LIN {X 0,Y 290.88,Z 169.752,A -85,B 0,C 180,E1 -16935.017,E2 -16935.017} C_VEL
LIN {X 0,Y 287.972,Z 170.097,A -85,B 0,C 180,E1 -16936.892,E2 -16936.892} C_VEL
LIN {X 0,Y 285.493,Z 170.39,A -85,B 0,C 180,E1 -16938.414,E2 -16938.414} C_VEL
LIN {X 0,Y 284.452,Z 170.52,A -85,B 0,C 180,E1 -16939.596,E2 -16939.596} C_VEL
LIN {X 0,Y 284.382,Z 170.533,A -85,B 0,C 180,E1 -16939.996,E2 -16939.996} C_VEL
LIN {X 0,Y 284.369,Z 170.558,A -85,B 0,C 180,E1 -16943.876,E2 -16943.876} C_VEL
LIN {X 0,Y 284.395,Z 170.53,A -85,B 0,C 180,E1 -16947.174,E2 -16947.174} C_VEL
LIN {X 0,Y 284.293,Z 170.571,A -85,B 0,C 180,E1 -16951.275,E2 -16951.275} C_VEL
LIN {X 0,Y 284.341,Z 170.55,A -85,B 0,C 180,E1 -16955.349,E2 -16955.349} C_VEL
LIN {X 0,Y 284.319,Z 170.568,A -85,B 0,C 180,E1 -16958.169,E2 -16958.169} C_VEL
LIN {X 0,Y 284.27,Z 170.574,A -85,B 0,C 180,E1 -16962.125,E2 -16962.125} C_VEL
LIN {X 0,Y 284.257,Z 170.577,A -85,B 0,C 180,E1 -16966.19,E2 -16966.19} C_VEL
LIN {X 0,Y 284.309,Z 170.539,A -85,B 0,C 180,E1 -16970.025,E2 -16970.025} C_VEL
LIN {X 0,Y 284.377,Z 170.673,A -85,B 0,C 180,E1 -16973.511,E2 -16973.511} C_VEL
LIN {X 0,Y 286.09,Z 178.895,A -85,B 0,C 180,E1 -16977.286,E2 -16977.286} C_VEL
LIN {X 0,Y 287.859,Z 188.158,A -85,B 0,C 180,E1 -16981.346,E2 -16981.346} C_VEL
LIN {X 0,Y 288.12,Z 189.357,A -85,B 0,C 180,E1 -16981.632,E2 -16981.632} C_VEL
LIN {X 0,Y 290.426,Z 195.694,A -85,B 0,C 180,E1 -16982.073,E2 -16982.073} C_VEL
LIN {X 0,Y 295.176,Z 217.529,A -85,B 0,C 180,E1 -16983.141,E2 -16983.141} C_VEL
LIN {X 0,Y 298.276,Z 235.786,A -85,B 0,C 180,E1 -16983.919,E2 -16983.919} C_VEL
LIN {X 0,Y 296.617,Z 295.017,A -85,B 0,C 180,E1 -16985.364,E2 -16985.364} C_VEL
LIN {X 0,Y 295.946,Z 305.327,A -85,B 0,C 180,E1 -16985.771,E2 -16985.771} C_VEL
LIN {X 0,Y 295.071,Z 314.839,A -85,B 0,C 180,E1 -16986.302,E2 -16986.302} C_VEL
LIN {X 0,Y 293.886,Z 324.916,A -85,B 0,C 180,E1 -16987.04,E2 -16987.04} C_VEL
LIN {X 0,Y 292.65,Z 334.674,A -85,B 0,C 180,E1 -16987.961,E2 -16987.961} C_VEL
LIN {X 0,Y 291.052,Z 344.737,A -85,B 0,C 180,E1 -16989.135,E2 -16989.135} C_VEL
LIN {X 0,Y 289.074,Z 356.234,A -85,B 0,C 180,E1 -16990.84,E2 -16990.84} C_VEL
LIN {X 0,Y 287.646,Z 364.301,A -85,B 0,C 180,E1 -16992.343,E2 -16992.343} C_VEL
LIN {X 0,Y 286.356,Z 371.575,A -85,B 0,C 180,E1 -16993.972,E2 -16993.972} C_VEL
LIN {X 0,Y 285.164,Z 378.112,A -85,B 0,C 180,E1 -16995.732,E2 -16995.732} C_VEL
LIN {X 0,Y 284.291,Z 382.612,A -85,B 0,C 180,E1 -16997.145,E2 -16997.145} C_VEL
LIN {X 0,Y 283.419,Z 388.106,A -85,B 0,C 180,E1 -16999.282,E2 -16999.282} C_VEL
LIN {X 0,Y 282.805,Z 392.433,A -85,B 0,C 180,E1 -17001.425,E2 -17001.425} C_VEL
LIN {X 0,Y 282.557,Z 394.802,A -85,B 0,C 180,E1 -17002.856,E2 -17002.856} C_VEL
LIN {X 0,Y 282.364,Z 397.026,A -85,B 0,C 180,E1 -17004.626,E2 -17004.626} C_VEL
LIN {X 0,Y 282.338,Z 399.054,A -85,B 0,C 180,E1 -17007.146,E2 -17007.146} C_VEL
LIN {X 0,Y 282.332,Z 399.644,A -85,B 0,C 180,E1 -17008.574,E2 -17008.574} C_VEL
LIN {X 0,Y 282.332,Z 399.644,A -85,B 0,C 180,E1 -17011.426,E2 -17011.426} C_VEL
LIN {X 0,Y 282.337,Z 399.054,A -85,B 0,C 180,E1 -17012.854,E2 -17012.854} C_VEL
LIN {X 0,Y 282.387,Z 396.602,A -85,B 0,C 180,E1 -17015.713,E2 -17015.713} C_VEL
LIN {X 0,Y 282.676,Z 393.651,A -85,B 0,C 180,E1 -17017.859,E2 -17017.859} C_VEL
LIN {X 0,Y 283.172,Z 389.66,A -85,B 0,C 180,E1 -17020.005,E2 -17020.005} C_VEL
LIN {X 0,Y 283.96,Z 384.528,A -85,B 0,C 180,E1 -17022.144,E2 -17022.144} C_VEL
LIN {X 0,Y 284.958,Z 379.268,A -85,B 0,C 180,E1 -17023.914,E2 -17023.914} C_VEL
LIN {X 0,Y 286.097,Z 372.951,A -85,B 0,C 180,E1 -17025.677,E2 -17025.677} C_VEL
LIN {X 0,Y 287.263,Z 367.002,A -85,B 0,C 180,E1 -17027.073,E2 -17027.073} C_VEL
LIN {X 0,Y 288.4,Z 360.072,A -85,B 0,C 180,E1 -17028.469,E2 -17028.469} C_VEL
LIN {X 0,Y 289.832,Z 351.895,A -85,B 0,C 180,E1 -17029.845,E2 -17029.845} C_VEL
LIN {X 0,Y 291.276,Z 343.386,A -85,B 0,C 180,E1 -17031.033,E2 -17031.033} C_VEL
LIN {X 0,Y 292.597,Z 334.673,A -85,B 0,C 180,E1 -17032.043,E2 -17032.043} C_VEL
LIN {X 0,Y 293.956,Z 324.918,A -85,B 0,C 180,E1 -17032.955,E2 -17032.955} C_VEL
LIN {X 0,Y 295.044,Z 314.838,A -85,B 0,C 180,E1 -17033.701,E2 -17033.701} C_VEL
LIN {X 0,Y 295.936,Z 305.326,A -85,B 0,C 180,E1 -17034.23,E2 -17034.23} C_VEL
LIN {X 0,Y 296.643,Z 295.017,A -85,B 0,C 180,E1 -17034.634,E2 -17034.634} C_VEL
LIN {X 0,Y 298.183,Z 234.871,A -85,B 0,C 180,E1 -17036.113,E2 -17036.113} C_VEL
LIN {X 0,Y 294.305,Z 213.339,A -85,B 0,C 180,E1 -17037.056,E2 -17037.056} C_VEL
LIN {X 0,Y 290.089,Z 194.522,A -85,B 0,C 180,E1 -17037.994,E2 -17037.994} C_VEL
LIN {X 0,Y 288.05,Z 189.055,A -85,B 0,C 180,E1 -17038.402,E2 -17038.402} C_VEL
LIN {X 0,Y 287.273,Z 184.811,A -85,B 0,C 180,E1 -17040.1,E2 -17040.1} C_VEL
LIN {X 0,Y 285.624,Z 176.503,A -85,B 0,C 180,E1 -17043.786,E2 -17043.786} C_VEL
LIN {X 0,Y 284.366,Z 170.578,A -85,B 0,C 180,E1 -17046.601,E2 -17046.601} C_VEL
LIN {X 0,Y 284.308,Z 170.539,A -85,B 0,C 180,E1 -17049.994,E2 -17049.994} C_VEL
LIN {X 0,Y 284.247,Z 170.575,A -85,B 0,C 180,E1 -17054.19,E2 -17054.19} C_VEL
LIN {X 0,Y 284.273,Z 170.574,A -85,B 0,C 180,E1 -17058.124,E2 -17058.124} C_VEL
LIN {X 0,Y 284.327,Z 170.567,A -85,B 0,C 180,E1 -17062.276,E2 -17062.276} C_VEL
LIN {X 0,Y 284.308,Z 170.548,A -85,B 0,C 180,E1 -17065.35,E2 -17065.35} C_VEL
LIN {X 0,Y 284.293,Z 170.571,A -85,B 0,C 180,E1 -17068.725,E2 -17068.725} C_VEL
LIN {X 0,Y 284.395,Z 170.53,A -85,B 0,C 180,E1 -17072.826,E2 -17072.826} C_VEL
LIN {X 0,Y 284.366,Z 170.561,A -85,B 0,C 180,E1 -17076.706,E2 -17076.706} C_VEL
LIN {X 0,Y 284.401,Z 170.521,A -85,B 0,C 180,E1 -17081.261,E2 -17081.261} C_VEL
LIN {X 0,Y 284.491,Z 170.539,A -85,B 0,C 180,E1 -17084.458,E2 -17084.458} C_VEL
LIN {X 0,Y 284.486,Z 170.522,A -85,B 0,C 180,E1 -17088.601,E2 -17088.601} C_VEL
LIN {X 0,Y 284.637,Z 170.496,A -85,B 0,C 180,E1 -17091.48,E2 -17091.48} C_VEL
LIN {X 0,Y 284.596,Z 170.532,A -85,B 0,C 180,E1 -17094.33,E2 -17094.33} C_VEL
LIN {X 0,Y 284.852,Z 170.475,A -85,B 0,C 180,E1 -17098.585,E2 -17098.585} C_VEL
LIN {X 0,Y 284.853,Z 170.47,A -85,B 0,C 180,E1 -17101.413,E2 -17101.413} C_VEL
LIN {X 0,Y 284.696,Z 170.513,A -85,B 0,C 180,E1 -17107.089,E2 -17107.089} C_VEL
LIN {X 0,Y 284.563,Z 170.5,A -85,B 0,C 180,E1 -17109.955,E2 -17109.955} C_VEL
LIN {X 0,Y 284.478,Z 170.55,A -85,B 0,C 180,E1 -17114.302,E2 -17114.302} C_VEL
LIN {X 0,Y 284.422,Z 170.536,A -85,B 0,C 180,E1 -17117.248,E2 -17117.248} C_VEL
LIN {X 0,Y 284.375,Z 170.533,A -85,B 0,C 180,E1 -17120.242,E2 -17120.242} C_VEL
LIN {X 0,Y 284.366,Z 170.563,A -85,B 0,C 180,E1 -17123.875,E2 -17123.875} C_VEL
LIN {X 0,Y 284.393,Z 170.531,A -85,B 0,C 180,E1 -17127.173,E2 -17127.173} C_VEL
LIN {X 0,Y 284.292,Z 170.575,A -85,B 0,C 180,E1 -17131.274,E2 -17131.274} C_VEL
LIN {X 0,Y 284.357,Z 170.544,A -85,B 0,C 180,E1 -17135.353,E2 -17135.353} C_VEL
LIN {X 0,Y 284.319,Z 170.569,A -85,B 0,C 180,E1 -17138.167,E2 -17138.167} C_VEL
LIN {X 0,Y 284.265,Z 170.569,A -85,B 0,C 180,E1 -17142.124,E2 -17142.124} C_VEL
LIN {X 0,Y 284.264,Z 170.535,A -85,B 0,C 180,E1 -17146.191,E2 -17146.191} C_VEL
LIN {X 0,Y 284.303,Z 170.538,A -85,B 0,C 180,E1 -17150.024,E2 -17150.024} C_VEL
LIN {X 0,Y 284.346,Z 170.546,A -85,B 0,C 180,E1 -17153.617,E2 -17153.617} C_VEL
LIN {X 0,Y 284.305,Z 170.553,A -85,B 0,C 180,E1 -17157.189,E2 -17157.189} C_VEL
LIN {X 0,Y 284.362,Z 170.704,A -85,B 0,C 180,E1 -17160.852,E2 -17160.852} C_VEL
LIN {X 0,Y 284.575,Z 171.612,A -85,B 0,C 180,E1 -17161.125,E2 -17161.125} C_VEL
LIN {X 0,Y 292.693,Z 186.861,A -85,B 0,C 180,E1 -17162.447,E2 -17162.447} C_VEL
LIN {X 0,Y 300.723,Z 198.195,A -85,B 0,C 180,E1 -17163.545,E2 -17163.545} C_VEL
LIN {X 0,Y 308.771,Z 207.249,A -85,B 0,C 180,E1 -17164.599,E2 -17164.599} C_VEL
LIN {X 0,Y 315.653,Z 214.555,A -85,B 0,C 180,E1 -17165.617,E2 -17165.617} C_VEL
LIN {X 0,Y 321.435,Z 220.417,A -85,B 0,C 180,E1 -17166.56,E2 -17166.56} C_VEL
LIN {X 0,Y 328.774,Z 227.475,A -85,B 0,C 180,E1 -17167.909,E2 -17167.909} C_VEL
LIN {X 0,Y 335.567,Z 233.937,A -85,B 0,C 180,E1 -17169.296,E2 -17169.296} C_VEL
LIN {X 0,Y 343.566,Z 240.897,A -85,B 0,C 180,E1 -17171.056,E2 -17171.056} C_VEL
LIN {X 0,Y 349.047,Z 245.344,A -85,B 0,C 180,E1 -17172.381,E2 -17172.381} C_VEL
LIN {X 0,Y 354.863,Z 250.07,A -85,B 0,C 180,E1 -17173.931,E2 -17173.931} C_VEL
LIN {X 0,Y 359.024,Z 253.254,A -85,B 0,C 180,E1 -17175.137,E2 -17175.137} C_VEL
LIN {X 0,Y 364.017,Z 257.245,A -85,B 0,C 180,E1 -17176.739,E2 -17176.739} C_VEL
LIN {X 0,Y 368.789,Z 260.213,A -85,B 0,C 180,E1 -17178.465,E2 -17178.465} C_VEL
LIN {X 0,Y 370.688,Z 261.609,A -85,B 0,C 180,E1 -17179.248,E2 -17179.248} C_VEL
LIN {X 0,Y 374.455,Z 264.816,A -85,B 0,C 180,E1 -17181.025,E2 -17181.025} C_VEL
LIN {X 0,Y 377.636,Z 266.924,A -85,B 0,C 180,E1 -17182.836,E2 -17182.836} C_VEL
LIN {X 0,Y 380.183,Z 268.235,A -85,B 0,C 180,E1 -17184.697,E2 -17184.697} C_VEL
LIN {X 0,Y 381.337,Z 268.729,A -85,B 0,C 180,E1 -17185.772,E2 -17185.772} C_VEL
LIN {X 0,Y 382.556,Z 269.148,A -85,B 0,C 180,E1 -17187.355,E2 -17187.355} C_VEL
LIN {X 0,Y 383.208,Z 269.566,A -85,B 0,C 180,E1 -17188.949,E2 -17188.949} C_VEL
LIN {X 0,Y 383.351,Z 269.507,A -85,B 0,C 180,E1 -17190,E2 -17190} C_VEL
LIN {X 0,Y 383.05,Z 269.43,A -85,B 0,C 180,E1 -17191.577,E2 -17191.577} C_VEL
LIN {X 0,Y 382.228,Z 268.951,A -85,B 0,C 180,E1 -17193.162,E2 -17193.162} C_VEL
LIN {X 0,Y 380.501,Z 268.419,A -85,B 0,C 180,E1 -17195.024,E2 -17195.024} C_VEL
LIN {X 0,Y 377.945,Z 267.115,A -85,B 0,C 180,E1 -17196.961,E2 -17196.961} C_VEL
LIN {X 0,Y 374.474,Z 264.83,A -85,B 0,C 180,E1 -17198.966,E2 -17198.966} C_VEL
LIN {X 0,Y 370.839,Z 261.73,A -85,B 0,C 180,E1 -17200.689,E2 -17200.689} C_VEL
LIN {X 0,Y 368.619,Z 260.105,A -85,B 0,C 180,E1 -17201.604,E2 -17201.604} C_VEL
LIN {X 0,Y 364.035,Z 257.251,A -85,B 0,C 180,E1 -17203.255,E2 -17203.255} C_VEL
LIN {X 0,Y 359.029,Z 253.234,A -85,B 0,C 180,E1 -17204.863,E2 -17204.863} C_VEL
LIN {X 0,Y 353.786,Z 249.277,A -85,B 0,C 180,E1 -17206.371,E2 -17206.371} C_VEL
LIN {X 0,Y 348.293,Z 244.643,A -85,B 0,C 180,E1 -17207.809,E2 -17207.809} C_VEL
LIN {X 0,Y 341.138,Z 238.842,A -85,B 0,C 180,E1 -17209.493,E2 -17209.493} C_VEL
LIN {X 0,Y 335.159,Z 233.574,A -85,B 0,C 180,E1 -17210.79,E2 -17210.79} C_VEL
LIN {X 0,Y 329.509,Z 228.106,A -85,B 0,C 180,E1 -17211.947,E2 -17211.947} C_VEL
LIN {X 0,Y 322.949,Z 221.914,A -85,B 0,C 180,E1 -17213.17,E2 -17213.17} C_VEL
LIN {X 0,Y 316.392,Z 215.413,A -85,B 0,C 180,E1 -17214.263,E2 -17214.263} C_VEL
LIN {X 0,Y 308.197,Z 206.704,A -85,B 0,C 180,E1 -17215.476,E2 -17215.476} C_VEL
LIN {X 0,Y 299.593,Z 196.708,A -85,B 0,C 180,E1 -17216.602,E2 -17216.602} C_VEL
LIN {X 0,Y 292.262,Z 186.12,A -85,B 0,C 180,E1 -17217.618,E2 -17217.618} C_VEL
LIN {X 0,Y 284.576,Z 171.61,A -85,B 0,C 180,E1 -17218.876,E2 -17218.876} C_VEL
LIN {X 0,Y 284.353,Z 170.626,A -85,B 0,C 180,E1 -17219.19,E2 -17219.19} C_VEL
LIN {X 0,Y 284.303,Z 170.551,A -85,B 0,C 180,E1 -17222.945,E2 -17222.945} C_VEL
LIN {X 0,Y 284.346,Z 170.546,A -85,B 0,C 180,E1 -17226.383,E2 -17226.383} C_VEL
LIN {X 0,Y 284.302,Z 170.537,A -85,B 0,C 180,E1 -17229.995,E2 -17229.995} C_VEL
LIN {X 0,Y 284.261,Z 170.543,A -85,B 0,C 180,E1 -17234.195,E2 -17234.195} C_VEL
LIN {X 0,Y 284.268,Z 170.565,A -85,B 0,C 180,E1 -17238.125,E2 -17238.125} C_VEL
LIN {X 0,Y 284.331,Z 170.57,A -85,B 0,C 180,E1 -17242.275,E2 -17242.275} C_VEL
LIN {X 0,Y 284.319,Z 170.544,A -85,B 0,C 180,E1 -17245.353,E2 -17245.353} C_VEL
LIN {X 0,Y 284.292,Z 170.575,A -85,B 0,C 180,E1 -17248.726,E2 -17248.726} C_VEL
LIN {X 0,Y 284.393,Z 170.531,A -85,B 0,C 180,E1 -17252.827,E2 -17252.827} C_VEL
LIN {X 0,Y 284.363,Z 170.563,A -85,B 0,C 180,E1 -17256.708,E2 -17256.708} C_VEL
LIN {X 0,Y 284.399,Z 170.523,A -85,B 0,C 180,E1 -17261.262,E2 -17261.262} C_VEL
LIN {X 0,Y 284.489,Z 170.547,A -85,B 0,C 180,E1 -17264.46,E2 -17264.46} C_VEL
LIN {X 0,Y 284.485,Z 170.522,A -85,B 0,C 180,E1 -17268.602,E2 -17268.602} C_VEL
LIN {X 0,Y 284.657,Z 170.498,A -85,B 0,C 180,E1 -17271.482,E2 -17271.482} C_VEL
LIN {X 0,Y 284.599,Z 170.534,A -85,B 0,C 180,E1 -17274.332,E2 -17274.332} C_VEL
LIN {X 0,Y 284.853,Z 170.47,A -85,B 0,C 180,E1 -17278.587,E2 -17278.587} C_VEL
LIN {X 0,Y 284.852,Z 170.475,A -85,B 0,C 180,E1 -17281.415,E2 -17281.415} C_VEL
LIN {X 0,Y 284.685,Z 170.508,A -85,B 0,C 180,E1 -17287.091,E2 -17287.091} C_VEL
LIN {X 0,Y 284.517,Z 170.505,A -85,B 0,C 180,E1 -17289.958,E2 -17289.958} C_VEL
LIN {X 0,Y 284.48,Z 170.545,A -85,B 0,C 180,E1 -17294.304,E2 -17294.304} C_VEL
LIN {X 0,Y 284.424,Z 170.529,A -85,B 0,C 180,E1 -17297.249,E2 -17297.249} C_VEL
LIN {X 0,Y 284.382,Z 170.533,A -85,B 0,C 180,E1 -17299.996,E2 -17299.996} C_VEL
LIN {X 0,Y 283.743,Z 170.628,A -85,B 0,C 180,E1 -17301.179,E2 -17301.179} C_VEL
LIN {X 0,Y 280.866,Z 170.999,A -85,B 0,C 180,E1 -17303.104,E2 -17303.104} C_VEL
LIN {X 0,Y 278.415,Z 171.293,A -85,B 0,C 180,E1 -17304.669,E2 -17304.669} C_VEL
LIN {X 0,Y 277.379,Z 171.409,A -85,B 0,C 180,E1 -17305.882,E2 -17305.882} C_VEL
LIN {X 0,Y 277.306,Z 171.414,A -85,B 0,C 180,E1 -17306.293,E2 -17306.293} C_VEL
LIN {X 0,Y 277.272,Z 171.447,A -85,B 0,C 180,E1 -17310.482,E2 -17310.482} C_VEL
LIN {X 0,Y 277.247,Z 171.426,A -85,B 0,C 180,E1 -17313.897,E2 -17313.897} C_VEL
LIN {X 0,Y 277.272,Z 171.447,A -85,B 0,C 180,E1 -17317.469,E2 -17317.469} C_VEL
LIN {X 0,Y 277.21,Z 171.445,A -85,B 0,C 180,E1 -17321.237,E2 -17321.237} C_VEL
LIN {X 0,Y 277.202,Z 171.447,A -85,B 0,C 180,E1 -17325.227,E2 -17325.227} C_VEL
LIN {X 0,Y 277.224,Z 171.421,A -85,B 0,C 180,E1 -17329.513,E2 -17329.513} C_VEL
LIN {X 0,Y 277.359,Z 171.598,A -85,B 0,C 180,E1 -17332.962,E2 -17332.962} C_VEL
LIN {X 0,Y 278.83,Z 178.676,A -85,B 0,C 180,E1 -17336.323,E2 -17336.323} C_VEL
LIN {X 0,Y 280.375,Z 186.527,A -85,B 0,C 180,E1 -17339.912,E2 -17339.912} C_VEL
LIN {X 0,Y 280.83,Z 188.826,A -85,B 0,C 180,E1 -17340.795,E2 -17340.795} C_VEL
LIN {X 0,Y 284.482,Z 198.321,A -85,B 0,C 180,E1 -17341.516,E2 -17341.516} C_VEL
LIN {X 0,Y 289.64,Z 223.006,A -85,B 0,C 180,E1 -17342.739,E2 -17342.739} C_VEL
LIN {X 0,Y 291.878,Z 236.965,A -85,B 0,C 180,E1 -17343.34,E2 -17343.34} C_VEL
LIN {X 0,Y 290.182,Z 294.832,A -85,B 0,C 180,E1 -17344.779,E2 -17344.779} C_VEL
LIN {X 0,Y 289.491,Z 305.135,A -85,B 0,C 180,E1 -17345.195,E2 -17345.195} C_VEL
LIN {X 0,Y 288.568,Z 314.647,A -85,B 0,C 180,E1 -17345.734,E2 -17345.734} C_VEL
LIN {X 0,Y 287.513,Z 323.719,A -85,B 0,C 180,E1 -17346.405,E2 -17346.405} C_VEL
LIN {X 0,Y 286.342,Z 332.852,A -85,B 0,C 180,E1 -17347.259,E2 -17347.259} C_VEL
LIN {X 0,Y 284.897,Z 341.844,A -85,B 0,C 180,E1 -17348.283,E2 -17348.283} C_VEL
LIN {X 0,Y 283.35,Z 350.568,A -85,B 0,C 180,E1 -17349.492,E2 -17349.492} C_VEL
LIN {X 0,Y 281.978,Z 357.96,A -85,B 0,C 180,E1 -17350.717,E2 -17350.717} C_VEL
LIN {X 0,Y 280.525,Z 366.236,A -85,B 0,C 180,E1 -17352.372,E2 -17352.372} C_VEL
LIN {X 0,Y 279.224,Z 372.758,A -85,B 0,C 180,E1 -17353.927,E2 -17353.927} C_VEL
LIN {X 0,Y 278.022,Z 379.075,A -85,B 0,C 180,E1 -17355.732,E2 -17355.732} C_VEL
LIN {X 0,Y 276.983,Z 384.336,A -85,B 0,C 180,E1 -17357.545,E2 -17357.545} C_VEL
LIN {X 0,Y 276.164,Z 389.468,A -85,B 0,C 180,E1 -17359.739,E2 -17359.739} C_VEL
LIN {X 0,Y 275.606,Z 393.458,A -85,B 0,C 180,E1 -17361.938,E2 -17361.938} C_VEL
LIN {X 0,Y 275.256,Z 397.09,A -85,B 0,C 180,E1 -17364.736,E2 -17364.736} C_VEL
LIN {X 0,Y 275.247,Z 398.862,A -85,B 0,C 180,E1 -17367.073,E2 -17367.073} C_VEL
LIN {X 0,Y 275.256,Z 399.453,A -85,B 0,C 180,E1 -17368.537,E2 -17368.537} C_VEL
LIN {X 0,Y 275.256,Z 399.453,A -85,B 0,C 180,E1 -17371.463,E2 -17371.463} C_VEL
LIN {X 0,Y 275.246,Z 398.862,A -85,B 0,C 180,E1 -17372.927,E2 -17372.927} C_VEL
LIN {X 0,Y 275.3,Z 396.41,A -85,B 0,C 180,E1 -17375.861,E2 -17375.861} C_VEL
LIN {X 0,Y 275.606,Z 393.458,A -85,B 0,C 180,E1 -17378.062,E2 -17378.062} C_VEL
LIN {X 0,Y 276.164,Z 389.468,A -85,B 0,C 180,E1 -17380.261,E2 -17380.261} C_VEL
LIN {X 0,Y 276.983,Z 384.336,A -85,B 0,C 180,E1 -17382.455,E2 -17382.455} C_VEL
LIN {X 0,Y 278.023,Z 379.075,A -85,B 0,C 180,E1 -17384.268,E2 -17384.268} C_VEL
LIN {X 0,Y 279.228,Z 372.758,A -85,B 0,C 180,E1 -17386.073,E2 -17386.073} C_VEL
LIN {X 0,Y 280.666,Z 365.808,A -85,B 0,C 180,E1 -17387.718,E2 -17387.718} C_VEL
LIN {X 0,Y 281.662,Z 359.88,A -85,B 0,C 180,E1 -17388.927,E2 -17388.927} C_VEL
LIN {X 0,Y 283.143,Z 351.702,A -85,B 0,C 180,E1 -17390.334,E2 -17390.334} C_VEL
LIN {X 0,Y 284.645,Z 343.194,A -85,B 0,C 180,E1 -17391.547,E2 -17391.547} C_VEL
LIN {X 0,Y 286.011,Z 334.481,A -85,B 0,C 180,E1 -17392.578,E2 -17392.578} C_VEL
LIN {X 0,Y 287.44,Z 324.727,A -85,B 0,C 180,E1 -17393.506,E2 -17393.506} C_VEL
LIN {X 0,Y 288.542,Z 314.646,A -85,B 0,C 180,E1 -17394.269,E2 -17394.269} C_VEL
LIN {X 0,Y 289.488,Z 305.135,A -85,B 0,C 180,E1 -17394.805,E2 -17394.805} C_VEL
LIN {X 0,Y 290.206,Z 294.826,A -85,B 0,C 180,E1 -17395.218,E2 -17395.218} C_VEL
LIN {X 0,Y 291.804,Z 235.968,A -85,B 0,C 180,E1 -17396.694,E2 -17396.694} C_VEL
LIN {X 0,Y 288.25,Z 215.924,A -85,B 0,C 180,E1 -17397.597,E2 -17397.597} C_VEL
LIN {X 0,Y 284.205,Z 197.401,A -85,B 0,C 180,E1 -17398.54,E2 -17398.54} C_VEL
LIN {X 0,Y 280.826,Z 188.828,A -85,B 0,C 180,E1 -17399.203,E2 -17399.203} C_VEL
LIN {X 0,Y 280.112,Z 185.125,A -85,B 0,C 180,E1 -17400.726,E2 -17400.726} C_VEL
LIN {X 0,Y 278.412,Z 176.684,A -85,B 0,C 180,E1 -17404.607,E2 -17404.607} C_VEL
LIN {X 0,Y 277.34,Z 171.483,A -85,B 0,C 180,E1 -17407.144,E2 -17407.144} C_VEL
LIN {X 0,Y 277.211,Z 171.427,A -85,B 0,C 180,E1 -17411.236,E2 -17411.236} C_VEL
LIN {X 0,Y 277.202,Z 171.446,A -85,B 0,C 180,E1 -17415.226,E2 -17415.226} C_VEL
LIN {X 0,Y 277.223,Z 171.438,A -85,B 0,C 180,E1 -17419.511,E2 -17419.511} C_VEL
LIN {X 0,Y 277.272,Z 171.447,A -85,B 0,C 180,E1 -17422.531,E2 -17422.531} C_VEL
LIN {X 0,Y 277.247,Z 171.426,A -85,B 0,C 180,E1 -17426.103,E2 -17426.103} C_VEL
LIN {X 0,Y 277.261,Z 171.448,A -85,B 0,C 180,E1 -17429.538,E2 -17429.538} C_VEL
LIN {X 0,Y 277.356,Z 171.406,A -85,B 0,C 180,E1 -17432.863,E2 -17432.863} C_VEL
LIN {X 0,Y 277.328,Z 171.435,A -85,B 0,C 180,E1 -17436.079,E2 -17436.079} C_VEL
LIN {X 0,Y 277.343,Z 171.401,A -85,B 0,C 180,E1 -17440.765,E2 -17440.765} C_VEL
LIN {X 0,Y 277.433,Z 171.424,A -85,B 0,C 180,E1 -17445.325,E2 -17445.325} C_VEL
LIN {X 0,Y 277.459,Z 171.384,A -85,B 0,C 180,E1 -17449.786,E2 -17449.786} C_VEL
LIN {X 0,Y 277.639,Z 171.383,A -85,B 0,C 180,E1 -17452.728,E2 -17452.728} C_VEL
LIN {X 0,Y 277.818,Z 171.351,A -85,B 0,C 180,E1 -17458.55,E2 -17458.55} C_VEL
LIN {X 0,Y 277.819,Z 171.346,A -85,B 0,C 180,E1 -17461.449,E2 -17461.449} C_VEL
LIN {X 0,Y 277.651,Z 171.387,A -85,B 0,C 180,E1 -17467.27,E2 -17467.27} C_VEL
LIN {X 0,Y 277.504,Z 171.379,A -85,B 0,C 180,E1 -17470.211,E2 -17470.211} C_VEL
LIN {X 0,Y 277.431,Z 171.426,A -85,B 0,C 180,E1 -17474.673,E2 -17474.673} C_VEL
LIN {X 0,Y 277.341,Z 171.401,A -85,B 0,C 180,E1 -17479.233,E2 -17479.233} C_VEL
LIN {X 0,Y 277.316,Z 171.439,A -85,B 0,C 180,E1 -17484.17,E2 -17484.17} C_VEL
LIN {X 0,Y 277.322,Z 171.412,A -85,B 0,C 180,E1 -17487.505,E2 -17487.505} C_VEL
LIN {X 0,Y 277.268,Z 171.447,A -85,B 0,C 180,E1 -17490.481,E2 -17490.481} C_VEL
LIN {X 0,Y 277.25,Z 171.426,A -85,B 0,C 180,E1 -17493.894,E2 -17493.894} C_VEL
LIN {X 0,Y 277.277,Z 171.449,A -85,B 0,C 180,E1 -17497.467,E2 -17497.467} C_VEL
LIN {X 0,Y 277.205,Z 171.438,A -85,B 0,C 180,E1 -17501.236,E2 -17501.236} C_VEL
LIN {X 0,Y 277.212,Z 171.434,A -85,B 0,C 180,E1 -17505.223,E2 -17505.223} C_VEL
LIN {X 0,Y 277.218,Z 171.408,A -85,B 0,C 180,E1 -17509.512,E2 -17509.512} C_VEL
LIN {X 0,Y 277.277,Z 171.445,A -85,B 0,C 180,E1 -17512.533,E2 -17512.533} C_VEL
LIN {X 0,Y 277.251,Z 171.416,A -85,B 0,C 180,E1 -17516.105,E2 -17516.105} C_VEL
LIN {X 0,Y 277.31,Z 171.569,A -85,B 0,C 180,E1 -17520.071,E2 -17520.071} C_VEL
LIN {X 0,Y 277.562,Z 172.52,A -85,B 0,C 180,E1 -17520.347,E2 -17520.347} C_VEL
LIN {X 0,Y 287.68,Z 191.464,A -85,B 0,C 180,E1 -17522.048,E2 -17522.048} C_VEL
LIN {X 0,Y 295.702,Z 202.853,A -85,B 0,C 180,E1 -17523.181,E2 -17523.181} C_VEL
LIN {X 0,Y 304.606,Z 212.79,A -85,B 0,C 180,E1 -17524.306,E2 -17524.306} C_VEL
LIN {X 0,Y 311.551,Z 220.017,A -85,B 0,C 180,E1 -17525.264,E2 -17525.264} C_VEL
LIN {X 0,Y 317.644,Z 226.073,A -85,B 0,C 180,E1 -17526.194,E2 -17526.194} C_VEL
LIN {X 0,Y 324.684,Z 232.783,A -85,B 0,C 180,E1 -17527.414,E2 -17527.414} C_VEL
LIN {X 0,Y 332.649,Z 240.066,A -85,B 0,C 180,E1 -17528.951,E2 -17528.951} C_VEL
LIN {X 0,Y 340.893,Z 247.172,A -85,B 0,C 180,E1 -17530.724,E2 -17530.724} C_VEL
LIN {X 0,Y 346.573,Z 251.663,A -85,B 0,C 180,E1 -17532.051,E2 -17532.051} C_VEL
LIN {X 0,Y 352.685,Z 256.556,A -85,B 0,C 180,E1 -17533.622,E2 -17533.622} C_VEL
LIN {X 0,Y 357.443,Z 260.17,A -85,B 0,C 180,E1 -17534.969,E2 -17534.969} C_VEL
LIN {X 0,Y 362.661,Z 264.181,A -85,B 0,C 180,E1 -17536.621,E2 -17536.621} C_VEL
LIN {X 0,Y 367.358,Z 267.075,A -85,B 0,C 180,E1 -17538.283,E2 -17538.283} C_VEL
LIN {X 0,Y 370.014,Z 269.137,A -85,B 0,C 180,E1 -17539.37,E2 -17539.37} C_VEL
LIN {X 0,Y 373.771,Z 272.138,A -85,B 0,C 180,E1 -17541.151,E2 -17541.151} C_VEL
LIN {X 0,Y 377.024,Z 274.168,A -85,B 0,C 180,E1 -17543.022,E2 -17543.022} C_VEL
LIN {X 0,Y 379.613,Z 275.436,A -85,B 0,C 180,E1 -17544.964,E2 -17544.964} C_VEL
LIN {X 0,Y 381.549,Z 276.095,A -85,B 0,C 180,E1 -17547.09,E2 -17547.09} C_VEL
LIN {X 0,Y 382.346,Z 276.596,A -85,B 0,C 180,E1 -17548.947,E2 -17548.947} C_VEL
LIN {X 0,Y 382.488,Z 276.539,A -85,B 0,C 180,E1 -17550,E2 -17550} C_VEL
LIN {X 0,Y 382.181,Z 276.479,A -85,B 0,C 180,E1 -17551.581,E2 -17551.581} C_VEL
LIN {X 0,Y 381.092,Z 275.929,A -85,B 0,C 180,E1 -17553.513,E2 -17553.513} C_VEL
LIN {X 0,Y 379.107,Z 275.218,A -85,B 0,C 180,E1 -17555.477,E2 -17555.477} C_VEL
LIN {X 0,Y 376.465,Z 273.808,A -85,B 0,C 180,E1 -17557.348,E2 -17557.348} C_VEL
LIN {X 0,Y 373.181,Z 271.695,A -85,B 0,C 180,E1 -17559.153,E2 -17559.153} C_VEL
LIN {X 0,Y 369.492,Z 268.668,A -85,B 0,C 180,E1 -17560.852,E2 -17560.852} C_VEL
LIN {X 0,Y 367.138,Z 266.937,A -85,B 0,C 180,E1 -17561.798,E2 -17561.798} C_VEL
LIN {X 0,Y 362.426,Z 264.047,A -85,B 0,C 180,E1 -17563.456,E2 -17563.456} C_VEL
LIN {X 0,Y 356.979,Z 259.754,A -85,B 0,C 180,E1 -17565.17,E2 -17565.17} C_VEL
LIN {X 0,Y 350.019,Z 254.576,A -85,B 0,C 180,E1 -17567.073,E2 -17567.073} C_VEL
LIN {X 0,Y 342.904,Z 248.679,A -85,B 0,C 180,E1 -17568.828,E2 -17568.828} C_VEL
LIN {X 0,Y 336.533,Z 243.402,A -85,B 0,C 180,E1 -17570.241,E2 -17570.241} C_VEL
LIN {X 0,Y 328.445,Z 236.331,A -85,B 0,C 180,E1 -17571.882,E2 -17571.882} C_VEL
LIN {X 0,Y 319.96,Z 228.31,A -85,B 0,C 180,E1 -17573.419,E2 -17573.419} C_VEL
LIN {X 0,Y 312.238,Z 220.798,A -85,B 0,C 180,E1 -17574.634,E2 -17574.634} C_VEL
LIN {X 0,Y 303.955,Z 212.169,A -85,B 0,C 180,E1 -17575.776,E2 -17575.776} C_VEL
LIN {X 0,Y 294.757,Z 201.562,A -85,B 0,C 180,E1 -17576.948,E2 -17576.948} C_VEL
LIN {X 0,Y 287.231,Z 190.721,A -85,B 0,C 180,E1 -17578.021,E2 -17578.021} C_VEL
LIN {X 0,Y 277.554,Z 172.541,A -85,B 0,C 180,E1 -17579.651,E2 -17579.651} C_VEL
LIN {X 0,Y 277.306,Z 171.517,A -85,B 0,C 180,E1 -17579.965,E2 -17579.965} C_VEL
LIN {X 0,Y 277.251,Z 171.416,A -85,B 0,C 180,E1 -17583.895,E2 -17583.895} C_VEL
LIN {X 0,Y 277.277,Z 171.445,A -85,B 0,C 180,E1 -17587.467,E2 -17587.467} C_VEL
LIN {X 0,Y 277.205,Z 171.401,A -85,B 0,C 180,E1 -17591.237,E2 -17591.237} C_VEL
LIN {X 0,Y 277.213,Z 171.442,A -85,B 0,C 180,E1 -17595.223,E2 -17595.223} C_VEL
LIN {X 0,Y 277.218,Z 171.435,A -85,B 0,C 180,E1 -17599.513,E2 -17599.513} C_VEL
LIN {X 0,Y 277.277,Z 171.449,A -85,B 0,C 180,E1 -17602.533,E2 -17602.533} C_VEL
LIN {X 0,Y 277.25,Z 171.426,A -85,B 0,C 180,E1 -17606.106,E2 -17606.106} C_VEL
LIN {X 0,Y 277.258,Z 171.449,A -85,B 0,C 180,E1 -17609.539,E2 -17609.539} C_VEL
LIN {X 0,Y 277.355,Z 171.407,A -85,B 0,C 180,E1 -17612.865,E2 -17612.865} C_VEL
LIN {X 0,Y 277.325,Z 171.439,A -85,B 0,C 180,E1 -17616.08,E2 -17616.08} C_VEL
LIN {X 0,Y 277.341,Z 171.401,A -85,B 0,C 180,E1 -17620.767,E2 -17620.767} C_VEL
LIN {X 0,Y 277.431,Z 171.426,A -85,B 0,C 180,E1 -17625.327,E2 -17625.327} C_VEL
LIN {X 0,Y 277.504,Z 171.379,A -85,B 0,C 180,E1 -17629.789,E2 -17629.789} C_VEL
LIN {X 0,Y 277.651,Z 171.387,A -85,B 0,C 180,E1 -17632.73,E2 -17632.73} C_VEL
LIN {X 0,Y 277.819,Z 171.346,A -85,B 0,C 180,E1 -17638.551,E2 -17638.551} C_VEL
LIN {X 0,Y 277.818,Z 171.351,A -85,B 0,C 180,E1 -17641.45,E2 -17641.45} C_VEL
LIN {X 0,Y 277.639,Z 171.383,A -85,B 0,C 180,E1 -17647.272,E2 -17647.272} C_VEL
LIN {X 0,Y 277.459,Z 171.384,A -85,B 0,C 180,E1 -17650.214,E2 -17650.214} C_VEL
LIN {X 0,Y 277.433,Z 171.424,A -85,B 0,C 180,E1 -17654.675,E2 -17654.675} C_VEL
LIN {X 0,Y 277.343,Z 171.401,A -85,B 0,C 180,E1 -17659.235,E2 -17659.235} C_VEL
LIN {X 0,Y 277.319,Z 171.436,A -85,B 0,C 180,E1 -17664.171,E2 -17664.171} C_VEL
LIN {X 0,Y 277.306,Z 171.414,A -85,B 0,C 180,E1 -17666.293,E2 -17666.293} C_VEL
LIN {X 0,Y 276.645,Z 171.499,A -85,B 0,C 180,E1 -17667.505,E2 -17667.505} C_VEL
LIN {X 0,Y 273.728,Z 171.882,A -85,B 0,C 180,E1 -17669.477,E2 -17669.477} C_VEL
LIN {X 0,Y 271.264,Z 172.195,A -85,B 0,C 180,E1 -17671.08,E2 -17671.08} C_VEL
LIN {X 0,Y 270.241,Z 172.312,A -85,B 0,C 180,E1 -17672.325,E2 -17672.325} C_VEL
LIN {X 0,Y 270.178,Z 172.312,A -85,B 0,C 180,E1 -17672.747,E2 -17672.747} C_VEL
LIN {X 0,Y 270.228,Z 172.322,A -85,B 0,C 180,E1 -17676.74,E2 -17676.74} C_VEL
LIN {X 0,Y 270.17,Z 172.319,A -85,B 0,C 180,E1 -17681.029,E2 -17681.029} C_VEL
LIN {X 0,Y 270.153,Z 172.326,A -85,B 0,C 180,E1 -17685.381,E2 -17685.381} C_VEL
LIN {X 0,Y 270.175,Z 172.298,A -85,B 0,C 180,E1 -17689.435,E2 -17689.435} C_VEL
LIN {X 0,Y 270.286,Z 172.466,A -85,B 0,C 180,E1 -17692.335,E2 -17692.335} C_VEL
LIN {X 0,Y 271.809,Z 179.574,A -85,B 0,C 180,E1 -17695.834,E2 -17695.834} C_VEL
LIN {X 0,Y 273.55,Z 188.467,A -85,B 0,C 180,E1 -17699.917,E2 -17699.917} C_VEL
LIN {X 0,Y 275.625,Z 193.635,A -85,B 0,C 180,E1 -17700.383,E2 -17700.383} C_VEL
LIN {X 0,Y 278.459,Z 200.725,A -85,B 0,C 180,E1 -17700.916,E2 -17700.916} C_VEL
LIN {X 0,Y 283.287,Z 223.884,A -85,B 0,C 180,E1 -17702.105,E2 -17702.105} C_VEL
LIN {X 0,Y 285.506,Z 237.888,A -85,B 0,C 180,E1 -17702.727,E2 -17702.727} C_VEL
LIN {X 0,Y 283.794,Z 294.647,A -85,B 0,C 180,E1 -17704.171,E2 -17704.171} C_VEL
LIN {X 0,Y 283.076,Z 304.944,A -85,B 0,C 180,E1 -17704.593,E2 -17704.593} C_VEL
LIN {X 0,Y 282.096,Z 314.454,A -85,B 0,C 180,E1 -17705.139,E2 -17705.139} C_VEL
LIN {X 0,Y 281.028,Z 323.527,A -85,B 0,C 180,E1 -17705.826,E2 -17705.826} C_VEL
LIN {X 0,Y 279.808,Z 332.66,A -85,B 0,C 180,E1 -17706.697,E2 -17706.697} C_VEL
LIN {X 0,Y 278.295,Z 341.652,A -85,B 0,C 180,E1 -17707.74,E2 -17707.74} C_VEL
LIN {X 0,Y 276.68,Z 350.376,A -85,B 0,C 180,E1 -17708.974,E2 -17708.974} C_VEL
LIN {X 0,Y 275.28,Z 357.768,A -85,B 0,C 180,E1 -17710.228,E2 -17710.228} C_VEL
LIN {X 0,Y 273.809,Z 365.316,A -85,B 0,C 180,E1 -17711.752,E2 -17711.752} C_VEL
LIN {X 0,Y 272.705,Z 371.19,A -85,B 0,C 180,E1 -17713.146,E2 -17713.146} C_VEL
LIN {X 0,Y 271.39,Z 377.728,A -85,B 0,C 180,E1 -17714.992,E2 -17714.992} C_VEL
LIN {X 0,Y 270.418,Z 382.228,A -85,B 0,C 180,E1 -17716.473,E2 -17716.473} C_VEL
LIN {X 0,Y 269.398,Z 387.721,A -85,B 0,C 180,E1 -17718.717,E2 -17718.717} C_VEL
LIN {X 0,Y 268.707,Z 392.048,A -85,B 0,C 180,E1 -17720.971,E2 -17720.971} C_VEL
LIN {X 0,Y 268.419,Z 394.417,A -85,B 0,C 180,E1 -17722.478,E2 -17722.478} C_VEL
LIN {X 0,Y 268.168,Z 397.069,A -85,B 0,C 180,E1 -17724.807,E2 -17724.807} C_VEL
LIN {X 0,Y 268.158,Z 398.67,A -85,B 0,C 180,E1 -17726.995,E2 -17726.995} C_VEL
LIN {X 0,Y 268.182,Z 399.262,A -85,B 0,C 180,E1 -17728.498,E2 -17728.498} C_VEL
LIN {X 0,Y 268.182,Z 399.262,A -85,B 0,C 180,E1 -17731.502,E2 -17731.502} C_VEL
LIN {X 0,Y 268.157,Z 398.67,A -85,B 0,C 180,E1 -17733.005,E2 -17733.005} C_VEL
LIN {X 0,Y 268.225,Z 396.218,A -85,B 0,C 180,E1 -17736.016,E2 -17736.016} C_VEL
LIN {X 0,Y 268.548,Z 393.266,A -85,B 0,C 180,E1 -17738.276,E2 -17738.276} C_VEL
LIN {X 0,Y 269.148,Z 389.276,A -85,B 0,C 180,E1 -17740.532,E2 -17740.532} C_VEL
LIN {X 0,Y 270.023,Z 384.143,A -85,B 0,C 180,E1 -17742.781,E2 -17742.781} C_VEL
LIN {X 0,Y 271.119,Z 378.883,A -85,B 0,C 180,E1 -17744.64,E2 -17744.64} C_VEL
LIN {X 0,Y 272.388,Z 372.566,A -85,B 0,C 180,E1 -17746.488,E2 -17746.488} C_VEL
LIN {X 0,Y 273.661,Z 366.617,A -85,B 0,C 180,E1 -17747.949,E2 -17747.949} C_VEL
LIN {X 0,Y 274.929,Z 359.688,A -85,B 0,C 180,E1 -17749.409,E2 -17749.409} C_VEL
LIN {X 0,Y 276.491,Z 351.511,A -85,B 0,C 180,E1 -17750.846,E2 -17750.846} C_VEL
LIN {X 0,Y 278.039,Z 343.002,A -85,B 0,C 180,E1 -17752.086,E2 -17752.086} C_VEL
LIN {X 0,Y 279.458,Z 334.289,A -85,B 0,C 180,E1 -17753.138,E2 -17753.138} C_VEL
LIN {X 0,Y 280.936,Z 324.535,A -85,B 0,C 180,E1 -17754.084,E2 -17754.084} C_VEL
LIN {X 0,Y 282.08,Z 314.454,A -85,B 0,C 180,E1 -17754.862,E2 -17754.862} C_VEL
LIN {X 0,Y 283.073,Z 304.944,A -85,B 0,C 180,E1 -17755.407,E2 -17755.407} C_VEL
LIN {X 0,Y 283.797,Z 294.634,A -85,B 0,C 180,E1 -17755.829,E2 -17755.829} C_VEL
LIN {X 0,Y 285.463,Z 237.191,A -85,B 0,C 180,E1 -17757.297,E2 -17757.297} C_VEL
LIN {X 0,Y 282.261,Z 218.578,A -85,B 0,C 180,E1 -17758.154,E2 -17758.154} C_VEL
LIN {X 0,Y 278.305,Z 200.083,A -85,B 0,C 180,E1 -17759.12,E2 -17759.12} C_VEL
LIN {X 0,Y 273.654,Z 188.866,A -85,B 0,C 180,E1 -17760.018,E2 -17760.018} C_VEL
LIN {X 0,Y 273.454,Z 188.003,A -85,B 0,C 180,E1 -17760.225,E2 -17760.225} C_VEL
LIN {X 0,Y 271.812,Z 179.571,A -85,B 0,C 180,E1 -17764.167,E2 -17764.167} C_VEL
LIN {X 0,Y 270.274,Z 172.351,A -85,B 0,C 180,E1 -17767.785,E2 -17767.785} C_VEL
LIN {X 0,Y 270.173,Z 172.324,A -85,B 0,C 180,E1 -17772.558,E2 -17772.558} C_VEL
LIN {X 0,Y 270.166,Z 172.332,A -85,B 0,C 180,E1 -17776.75,E2 -17776.75} C_VEL
LIN {X 0,Y 270.174,Z 172.316,A -85,B 0,C 180,E1 -17779.433,E2 -17779.433} C_VEL
LIN {X 0,Y 270.243,Z 172.317,A -85,B 0,C 180,E1 -17783.725,E2 -17783.725} C_VEL
LIN {X 0,Y 270.202,Z 172.308,A -85,B 0,C 180,E1 -17786.892,E2 -17786.892} C_VEL
LIN {X 0,Y 270.219,Z 172.322,A -85,B 0,C 180,E1 -17790.385,E2 -17790.385} C_VEL
LIN {X 0,Y 270.262,Z 172.291,A -85,B 0,C 180,E1 -17793.763,E2 -17793.763} C_VEL
LIN {X 0,Y 270.233,Z 172.323,A -85,B 0,C 180,E1 -17797.038,E2 -17797.038} C_VEL
LIN {X 0,Y 270.301,Z 172.282,A -85,B 0,C 180,E1 -17800.244,E2 -17800.244} C_VEL
LIN {X 0,Y 270.402,Z 172.298,A -85,B 0,C 180,E1 -17804.935,E2 -17804.935} C_VEL
LIN {X 0,Y 270.411,Z 172.263,A -85,B 0,C 180,E1 -17809.517,E2 -17809.517} C_VEL
LIN {X 0,Y 270.597,Z 172.257,A -85,B 0,C 180,E1 -17812.538,E2 -17812.538} C_VEL
LIN {X 0,Y 270.784,Z 172.226,A -85,B 0,C 180,E1 -17818.512,E2 -17818.512} C_VEL
LIN {X 0,Y 270.785,Z 172.221,A -85,B 0,C 180,E1 -17821.486,E2 -17821.486} C_VEL
LIN {X 0,Y 270.609,Z 172.26,A -85,B 0,C 180,E1 -17827.46,E2 -17827.46} C_VEL
LIN {X 0,Y 270.439,Z 172.259,A -85,B 0,C 180,E1 -17830.48,E2 -17830.48} C_VEL
LIN {X 0,Y 270.4,Z 172.302,A -85,B 0,C 180,E1 -17835.064,E2 -17835.064} C_VEL
LIN {X 0,Y 270.298,Z 172.28,A -85,B 0,C 180,E1 -17839.755,E2 -17839.755} C_VEL
LIN {X 0,Y 270.271,Z 172.315,A -85,B 0,C 180,E1 -17844.585,E2 -17844.585} C_VEL
LIN {X 0,Y 270.268,Z 172.291,A -85,B 0,C 180,E1 -17847.908,E2 -17847.908} C_VEL
LIN {X 0,Y 270.18,Z 172.333,A -85,B 0,C 180,E1 -17851.348,E2 -17851.348} C_VEL
LIN {X 0,Y 270.211,Z 172.302,A -85,B 0,C 180,E1 -17854.903,E2 -17854.903} C_VEL
LIN {X 0,Y 270.218,Z 172.323,A -85,B 0,C 180,E1 -17858.717,E2 -17858.717} C_VEL
LIN {X 0,Y 270.168,Z 172.334,A -85,B 0,C 180,E1 -17863.25,E2 -17863.25} C_VEL
LIN {X 0,Y 270.17,Z 172.273,A -85,B 0,C 180,E1 -17867.442,E2 -17867.442} C_VEL
LIN {X 0,Y 270.203,Z 172.324,A -85,B 0,C 180,E1 -17871.374,E2 -17871.374} C_VEL
LIN {X 0,Y 270.211,Z 172.289,A -85,B 0,C 180,E1 -17875.096,E2 -17875.096} C_VEL
LIN {X 0,Y 270.248,Z 172.541,A -85,B 0,C 180,E1 -17879.292,E2 -17879.292} C_VEL
LIN {X 0,Y 270.532,Z 173.631,A -85,B 0,C 180,E1 -17879.534,E2 -17879.534} C_VEL
LIN {X 0,Y 282.95,Z 196.514,A -85,B 0,C 180,E1 -17881.677,E2 -17881.677} C_VEL
LIN {X 0,Y 291.272,Z 208.222,A -85,B 0,C 180,E1 -17882.882,E2 -17882.882} C_VEL
LIN {X 0,Y 300.351,Z 218.305,A -85,B 0,C 180,E1 -17884.036,E2 -17884.036} C_VEL
LIN {X 0,Y 307.234,Z 225.317,A -85,B 0,C 180,E1 -17884.917,E2 -17884.917} C_VEL
LIN {X 0,Y 313.893,Z 231.833,A -85,B 0,C 180,E1 -17885.871,E2 -17885.871} C_VEL
LIN {X 0,Y 321.781,Z 239.116,A -85,B 0,C 180,E1 -17887.148,E2 -17887.148} C_VEL
LIN {X 0,Y 329.753,Z 246.296,A -85,B 0,C 180,E1 -17888.633,E2 -17888.633} C_VEL
LIN {X 0,Y 338.441,Z 253.613,A -85,B 0,C 180,E1 -17890.442,E2 -17890.442} C_VEL
LIN {X 0,Y 344.396,Z 258.326,A -85,B 0,C 180,E1 -17891.809,E2 -17891.809} C_VEL
LIN {X 0,Y 350.613,Z 263.151,A -85,B 0,C 180,E1 -17893.358,E2 -17893.358} C_VEL
LIN {X 0,Y 356.079,Z 267.284,A -85,B 0,C 180,E1 -17894.876,E2 -17894.876} C_VEL
LIN {X 0,Y 361.766,Z 271.468,A -85,B 0,C 180,E1 -17896.655,E2 -17896.655} C_VEL
LIN {X 0,Y 366.511,Z 274.236,A -85,B 0,C 180,E1 -17898.324,E2 -17898.324} C_VEL
LIN {X 0,Y 370.879,Z 277.818,A -85,B 0,C 180,E1 -17900.186,E2 -17900.186} C_VEL
LIN {X 0,Y 374.243,Z 280.136,A -85,B 0,C 180,E1 -17901.892,E2 -17901.892} C_VEL
LIN {X 0,Y 377.192,Z 281.782,A -85,B 0,C 180,E1 -17903.736,E2 -17903.736} C_VEL
LIN {X 0,Y 379.568,Z 282.788,A -85,B 0,C 180,E1 -17905.753,E2 -17905.753} C_VEL
LIN {X 0,Y 380.815,Z 283.242,A -85,B 0,C 180,E1 -17907.343,E2 -17907.343} C_VEL
LIN {X 0,Y 381.48,Z 283.642,A -85,B 0,C 180,E1 -17908.944,E2 -17908.944} C_VEL
LIN {X 0,Y 381.624,Z 283.577,A -85,B 0,C 180,E1 -17910,E2 -17910} C_VEL
LIN {X 0,Y 381.313,Z 283.519,A -85,B 0,C 180,E1 -17911.584,E2 -17911.584} C_VEL
LIN {X 0,Y 380.222,Z 282.958,A -85,B 0,C 180,E1 -17913.515,E2 -17913.515} C_VEL
LIN {X 0,Y 378.215,Z 282.263,A -85,B 0,C 180,E1 -17915.49,E2 -17915.49} C_VEL
LIN {X 0,Y 375.564,Z 280.908,A -85,B 0,C 180,E1 -17917.348,E2 -17917.348} C_VEL
LIN {X 0,Y 372.03,Z 278.678,A -85,B 0,C 180,E1 -17919.26,E2 -17919.26} C_VEL
LIN {X 0,Y 368.376,Z 275.808,A -85,B 0,C 180,E1 -17920.918,E2 -17920.918} C_VEL
LIN {X 0,Y 366.019,Z 273.983,A -85,B 0,C 180,E1 -17921.856,E2 -17921.856} C_VEL
LIN {X 0,Y 361.119,Z 271.047,A -85,B 0,C 180,E1 -17923.559,E2 -17923.559} C_VEL
LIN {X 0,Y 355.429,Z 266.724,A -85,B 0,C 180,E1 -17925.318,E2 -17925.318} C_VEL
LIN {X 0,Y 348.219,Z 261.412,A -85,B 0,C 180,E1 -17927.248,E2 -17927.248} C_VEL
LIN {X 0,Y 342.531,Z 256.639,A -85,B 0,C 180,E1 -17928.644,E2 -17928.644} C_VEL
LIN {X 0,Y 335.46,Z 251.169,A -85,B 0,C 180,E1 -17930.199,E2 -17930.199} C_VEL
LIN {X 0,Y 327.92,Z 244.775,A -85,B 0,C 180,E1 -17931.72,E2 -17931.72} C_VEL
LIN {X 0,Y 319.294,Z 236.938,A -85,B 0,C 180,E1 -17933.268,E2 -17933.268} C_VEL
LIN {X 0,Y 310.366,Z 228.579,A -85,B 0,C 180,E1 -17934.641,E2 -17934.641} C_VEL
LIN {X 0,Y 301.212,Z 219.269,A -85,B 0,C 180,E1 -17935.857,E2 -17935.857} C_VEL
LIN {X 0,Y 290.79,Z 207.568,A -85,B 0,C 180,E1 -17937.185,E2 -17937.185} C_VEL
LIN {X 0,Y 282.71,Z 196.115,A -85,B 0,C 180,E1 -17938.36,E2 -17938.36} C_VEL
LIN {X 0,Y 275.546,Z 182.971,A -85,B 0,C 180,E1 -17939.56,E2 -17939.56} C_VEL
LIN {X 0,Y 270.442,Z 173.384,A -85,B 0,C 180,E1 -17940.496,E2 -17940.496} C_VEL
LIN {X 0,Y 270.212,Z 172.414,A -85,B 0,C 180,E1 -17940.818,E2 -17940.818} C_VEL
LIN {X 0,Y 270.211,Z 172.289,A -85,B 0,C 180,E1 -17944.904,E2 -17944.904} C_VEL
LIN {X 0,Y 270.218,Z 172.321,A -85,B 0,C 180,E1 -17948.717,E2 -17948.717} C_VEL
LIN {X 0,Y 270.167,Z 172.279,A -85,B 0,C 180,E1 -17953.251,E2 -17953.251} C_VEL
LIN {X 0,Y 270.17,Z 172.329,A -85,B 0,C 180,E1 -17957.443,E2 -17957.443} C_VEL
LIN {X 0,Y 270.203,Z 172.326,A -85,B 0,C 180,E1 -17961.375,E2 -17961.375} C_VEL
LIN {X 0,Y 270.211,Z 172.302,A -85,B 0,C 180,E1 -17965.097,E2 -17965.097} C_VEL
LIN {X 0,Y 270.197,Z 172.329,A -85,B 0,C 180,E1 -17969.131,E2 -17969.131} C_VEL
LIN {X 0,Y 270.261,Z 172.292,A -85,B 0,C 180,E1 -17972.146,E2 -17972.146} C_VEL
LIN {X 0,Y 270.274,Z 172.314,A -85,B 0,C 180,E1 -17975.52,E2 -17975.52} C_VEL
LIN {X 0,Y 270.298,Z 172.28,A -85,B 0,C 180,E1 -17980.245,E2 -17980.245} C_VEL
LIN {X 0,Y 270.4,Z 172.302,A -85,B 0,C 180,E1 -17984.936,E2 -17984.936} C_VEL
LIN {X 0,Y 270.439,Z 172.259,A -85,B 0,C 180,E1 -17989.52,E2 -17989.52} C_VEL
LIN {X 0,Y 270.609,Z 172.26,A -85,B 0,C 180,E1 -17992.54,E2 -17992.54} C_VEL
LIN {X 0,Y 270.785,Z 172.221,A -85,B 0,C 180,E1 -17998.514,E2 -17998.514} C_VEL
LIN {X 0,Y 270.784,Z 172.226,A -85,B 0,C 180,E1 -18001.488,E2 -18001.488} C_VEL
LIN {X 0,Y 270.597,Z 172.257,A -85,B 0,C 180,E1 -18007.462,E2 -18007.462} C_VEL
LIN {X 0,Y 270.411,Z 172.263,A -85,B 0,C 180,E1 -18010.483,E2 -18010.483} C_VEL
LIN {X 0,Y 270.402,Z 172.298,A -85,B 0,C 180,E1 -18015.065,E2 -18015.065} C_VEL
LIN {X 0,Y 270.301,Z 172.282,A -85,B 0,C 180,E1 -18019.756,E2 -18019.756} C_VEL
LIN {X 0,Y 270.274,Z 172.308,A -85,B 0,C 180,E1 -18024.586,E2 -18024.586} C_VEL
LIN {X 0,Y 270.269,Z 172.293,A -85,B 0,C 180,E1 -18027.91,E2 -18027.91} C_VEL
LIN {X 0,Y 270.184,Z 172.328,A -85,B 0,C 180,E1 -18031.349,E2 -18031.349} C_VEL
LIN {X 0,Y 270.178,Z 172.312,A -85,B 0,C 180,E1 -18032.747,E2 -18032.747} C_VEL
LIN {X 0,Y 269.564,Z 172.389,A -85,B 0,C 180,E1 -18033.992,E2 -18033.992} C_VEL
LIN {X 0,Y 266.729,Z 172.752,A -85,B 0,C 180,E1 -18036.02,E2 -18036.02} C_VEL
LIN {X 0,Y 264.279,Z 173.065,A -85,B 0,C 180,E1 -18037.67,E2 -18037.67} C_VEL
LIN {X 0,Y 263.208,Z 173.188,A -85,B 0,C 180,E1 -18038.949,E2 -18038.949} C_VEL
LIN {X 0,Y 263.113,Z 173.196,A -85,B 0,C 180,E1 -18039.383,E2 -18039.383} C_VEL
LIN {X 0,Y 263.124,Z 173.207,A -85,B 0,C 180,E1 -18041.894,E2 -18041.894} C_VEL
LIN {X 0,Y 263.125,Z 173.209,A -85,B 0,C 180,E1 -18046.152,E2 -18046.152} C_VEL
LIN {X 0,Y 263.116,Z 173.177,A -85,B 0,C 180,E1 -18050.13,E2 -18050.13} C_VEL
LIN {X 0,Y 263.217,Z 173.286,A -85,B 0,C 180,E1 -18051.636,E2 -18051.636} C_VEL
LIN {X 0,Y 264.799,Z 180.569,A -85,B 0,C 180,E1 -18055.364,E2 -18055.364} C_VEL
LIN {X 0,Y 266.268,Z 188.153,A -85,B 0,C 180,E1 -18058.982,E2 -18058.982} C_VEL
LIN {X 0,Y 267.764,Z 191.843,A -85,B 0,C 180,E1 -18059.375,E2 -18059.375} C_VEL
LIN {X 0,Y 272.506,Z 203.241,A -85,B 0,C 180,E1 -18060.298,E2 -18060.298} C_VEL
LIN {X 0,Y 277.246,Z 226.307,A -85,B 0,C 180,E1 -18061.517,E2 -18061.517} C_VEL
LIN {X 0,Y 279.168,Z 238.832,A -85,B 0,C 180,E1 -18062.087,E2 -18062.087} C_VEL
LIN {X 0,Y 277.423,Z 294.462,A -85,B 0,C 180,E1 -18063.532,E2 -18063.532} C_VEL
LIN {X 0,Y 276.689,Z 304.753,A -85,B 0,C 180,E1 -18063.963,E2 -18063.963} C_VEL
LIN {X 0,Y 275.687,Z 314.263,A -85,B 0,C 180,E1 -18064.521,E2 -18064.521} C_VEL
LIN {X 0,Y 274.564,Z 323.336,A -85,B 0,C 180,E1 -18065.219,E2 -18065.219} C_VEL
LIN {X 0,Y 273.295,Z 332.468,A -85,B 0,C 180,E1 -18066.108,E2 -18066.108} C_VEL
LIN {X 0,Y 271.707,Z 341.459,A -85,B 0,C 180,E1 -18067.171,E2 -18067.171} C_VEL
LIN {X 0,Y 270.074,Z 350.184,A -85,B 0,C 180,E1 -18068.435,E2 -18068.435} C_VEL
LIN {X 0,Y 268.581,Z 357.576,A -85,B 0,C 180,E1 -18069.714,E2 -18069.714} C_VEL
LIN {X 0,Y 266.89,Z 365.855,A -85,B 0,C 180,E1 -18071.441,E2 -18071.441} C_VEL
LIN {X 0,Y 265.905,Z 371.018,A -85,B 0,C 180,E1 -18072.708,E2 -18072.708} C_VEL
LIN {X 0,Y 264.51,Z 377.535,A -85,B 0,C 180,E1 -18074.592,E2 -18074.592} C_VEL
LIN {X 0,Y 263.509,Z 382.036,A -85,B 0,C 180,E1 -18076.111,E2 -18076.111} C_VEL
LIN {X 0,Y 262.407,Z 387.528,A -85,B 0,C 180,E1 -18078.412,E2 -18078.412} C_VEL
LIN {X 0,Y 261.687,Z 391.856,A -85,B 0,C 180,E1 -18080.727,E2 -18080.727} C_VEL
LIN {X 0,Y 261.353,Z 394.225,A -85,B 0,C 180,E1 -18082.273,E2 -18082.273} C_VEL
LIN {X 0,Y 261.088,Z 397.029,A -85,B 0,C 180,E1 -18084.863,E2 -18084.863} C_VEL
LIN {X 0,Y 261.054,Z 398.478,A -85,B 0,C 180,E1 -18086.914,E2 -18086.914} C_VEL
LIN {X 0,Y 261.088,Z 399.07,A -85,B 0,C 180,E1 -18088.458,E2 -18088.458} C_VEL
LIN {X 0,Y 261.088,Z 399.07,A -85,B 0,C 180,E1 -18091.542,E2 -18091.542} C_VEL
LIN {X 0,Y 261.052,Z 398.478,A -85,B 0,C 180,E1 -18093.086,E2 -18093.086} C_VEL
LIN {X 0,Y 261.151,Z 396.026,A -85,B 0,C 180,E1 -18096.18,E2 -18096.18} C_VEL
LIN {X 0,Y 261.51,Z 393.074,A -85,B 0,C 180,E1 -18098.5,E2 -18098.5} C_VEL
LIN {X 0,Y 262.123,Z 389.083,A -85,B 0,C 180,E1 -18100.817,E2 -18100.817} C_VEL
LIN {X 0,Y 263.082,Z 383.951,A -85,B 0,C 180,E1 -18103.124,E2 -18103.124} C_VEL
LIN {X 0,Y 264.238,Z 378.69,A -85,B 0,C 180,E1 -18105.03,E2 -18105.03} C_VEL
LIN {X 0,Y 265.572,Z 372.374,A -85,B 0,C 180,E1 -18106.924,E2 -18106.924} C_VEL
LIN {X 0,Y 266.865,Z 366.424,A -85,B 0,C 180,E1 -18108.422,E2 -18108.422} C_VEL
LIN {X 0,Y 268.221,Z 359.496,A -85,B 0,C 180,E1 -18109.915,E2 -18109.915} C_VEL
LIN {X 0,Y 269.853,Z 351.319,A -85,B 0,C 180,E1 -18111.384,E2 -18111.384} C_VEL
LIN {X 0,Y 271.458,Z 342.81,A -85,B 0,C 180,E1 -18112.65,E2 -18112.65} C_VEL
LIN {X 0,Y 272.934,Z 334.097,A -85,B 0,C 180,E1 -18113.724,E2 -18113.724} C_VEL
LIN {X 0,Y 274.465,Z 324.344,A -85,B 0,C 180,E1 -18114.689,E2 -18114.689} C_VEL
LIN {X 0,Y 275.526,Z 315.55,A -85,B 0,C 180,E1 -18115.394,E2 -18115.394} C_VEL
LIN {X 0,Y 276.585,Z 305.626,A -85,B 0,C 180,E1 -18115.997,E2 -18115.997} C_VEL
LIN {X 0,Y 277.377,Z 295.775,A -85,B 0,C 180,E1 -18116.422,E2 -18116.422} C_VEL
LIN {X 0,Y 278.18,Z 270.277,A -85,B 0,C 180,E1 -18117.125,E2 -18117.125} C_VEL
LIN {X 0,Y 279.11,Z 238.02,A -85,B 0,C 180,E1 -18117.943,E2 -18117.943} C_VEL
LIN {X 0,Y 276.042,Z 220.052,A -85,B 0,C 180,E1 -18118.799,E2 -18118.799} C_VEL
LIN {X 0,Y 272.211,Z 202.241,A -85,B 0,C 180,E1 -18119.767,E2 -18119.767} C_VEL
LIN {X 0,Y 266.387,Z 188.582,A -85,B 0,C 180,E1 -18120.932,E2 -18120.932} C_VEL
LIN {X 0,Y 266.126,Z 187.394,A -85,B 0,C 180,E1 -18121.297,E2 -18121.297} C_VEL
LIN {X 0,Y 264.586,Z 179.647,A -85,B 0,C 180,E1 -18125.096,E2 -18125.096} C_VEL
LIN {X 0,Y 263.202,Z 173.219,A -85,B 0,C 180,E1 -18128.486,E2 -18128.486} C_VEL
LIN {X 0,Y 263.125,Z 173.188,A -85,B 0,C 180,E1 -18131.893,E2 -18131.893} C_VEL
LIN {X 0,Y 263.106,Z 173.205,A -85,B 0,C 180,E1 -18136.154,E2 -18136.154} C_VEL
LIN {X 0,Y 263.106,Z 173.195,A -85,B 0,C 180,E1 -18140.127,E2 -18140.127} C_VEL
LIN {X 0,Y 263.176,Z 173.194,A -85,B 0,C 180,E1 -18144.019,E2 -18144.019} C_VEL
LIN {X 0,Y 263.133,Z 173.198,A -85,B 0,C 180,E1 -18147.711,E2 -18147.711} C_VEL
LIN {X 0,Y 263.198,Z 173.176,A -85,B 0,C 180,E1 -18151.783,E2 -18151.783} C_VEL
LIN {X 0,Y 263.226,Z 173.183,A -85,B 0,C 180,E1 -18155.2,E2 -18155.2} C_VEL
LIN {X 0,Y 263.263,Z 173.165,A -85,B 0,C 180,E1 -18159.693,E2 -18159.693} C_VEL
LIN {X 0,Y 263.35,Z 173.173,A -85,B 0,C 180,E1 -18164.521,E2 -18164.521} C_VEL
LIN {X 0,Y 263.354,Z 173.144,A -85,B 0,C 180,E1 -18169.233,E2 -18169.233} C_VEL
LIN {X 0,Y 263.557,Z 173.132,A -85,B 0,C 180,E1 -18172.337,E2 -18172.337} C_VEL
LIN {X 0,Y 263.748,Z 173.102,A -85,B 0,C 180,E1 -18178.472,E2 -18178.472} C_VEL
LIN {X 0,Y 263.749,Z 173.097,A -85,B 0,C 180,E1 -18181.526,E2 -18181.526} C_VEL
LIN {X 0,Y 263.571,Z 173.132,A -85,B 0,C 180,E1 -18187.661,E2 -18187.661} C_VEL
LIN {X 0,Y 263.371,Z 173.141,A -85,B 0,C 180,E1 -18190.765,E2 -18190.765} C_VEL
LIN {X 0,Y 263.348,Z 173.18,A -85,B 0,C 180,E1 -18195.477,E2 -18195.477} C_VEL
LIN {X 0,Y 263.26,Z 173.161,A -85,B 0,C 180,E1 -18200.306,E2 -18200.306} C_VEL
LIN {X 0,Y 263.205,Z 173.185,A -85,B 0,C 180,E1 -18205.291,E2 -18205.291} C_VEL
LIN {X 0,Y 263.176,Z 173.182,A -85,B 0,C 180,E1 -18208.729,E2 -18208.729} C_VEL
LIN {X 0,Y 263.13,Z 173.205,A -85,B 0,C 180,E1 -18212.288,E2 -18212.288} C_VEL
LIN {X 0,Y 263.183,Z 173.187,A -85,B 0,C 180,E1 -18215.978,E2 -18215.978} C_VEL
LIN {X 0,Y 263.11,Z 173.194,A -85,B 0,C 180,E1 -18219.87,E2 -18219.87} C_VEL
LIN {X 0,Y 263.124,Z 173.207,A -85,B 0,C 180,E1 -18223.983,E2 -18223.983} C_VEL
LIN {X 0,Y 263.12,Z 173.15,A -85,B 0,C 180,E1 -18228.406,E2 -18228.406} C_VEL
LIN {X 0,Y 263.162,Z 173.207,A -85,B 0,C 180,E1 -18232.104,E2 -18232.104} C_VEL
LIN {X 0,Y 263.18,Z 173.165,A -85,B 0,C 180,E1 -18235.89,E2 -18235.89} C_VEL
LIN {X 0,Y 263.171,Z 173.408,A -85,B 0,C 180,E1 -18238.397,E2 -18238.397} C_VEL
LIN {X 0,Y 263.401,Z 174.364,A -85,B 0,C 180,E1 -18238.627,E2 -18238.627} C_VEL
LIN {X 0,Y 272.651,Z 191.663,A -85,B 0,C 180,E1 -18240.351,E2 -18240.351} C_VEL
LIN {X 0,Y 278.843,Z 202.423,A -85,B 0,C 180,E1 -18241.388,E2 -18241.388} C_VEL
LIN {X 0,Y 286.978,Z 213.718,A -85,B 0,C 180,E1 -18242.59,E2 -18242.59} C_VEL
LIN {X 0,Y 298.365,Z 226.339,A -85,B 0,C 180,E1 -18244.059,E2 -18244.059} C_VEL
LIN {X 0,Y 308.558,Z 236.264,A -85,B 0,C 180,E1 -18245.357,E2 -18245.357} C_VEL
LIN {X 0,Y 317.172,Z 244.082,A -85,B 0,C 180,E1 -18246.644,E2 -18246.644} C_VEL
LIN {X 0,Y 325.041,Z 251.035,A -85,B 0,C 180,E1 -18248.004,E2 -18248.004} C_VEL
LIN {X 0,Y 332.818,Z 257.588,A -85,B 0,C 180,E1 -18249.517,E2 -18249.517} C_VEL
LIN {X 0,Y 341.237,Z 264.116,A -85,B 0,C 180,E1 -18251.332,E2 -18251.332} C_VEL
LIN {X 0,Y 347.827,Z 269.272,A -85,B 0,C 180,E1 -18252.936,E2 -18252.936} C_VEL
LIN {X 0,Y 353.23,Z 273.209,A -85,B 0,C 180,E1 -18254.373,E2 -18254.373} C_VEL
LIN {X 0,Y 358.229,Z 276.979,A -85,B 0,C 180,E1 -18255.853,E2 -18255.853} C_VEL
LIN {X 0,Y 363.473,Z 280.279,A -85,B 0,C 180,E1 -18257.572,E2 -18257.572} C_VEL
LIN {X 0,Y 366.024,Z 281.791,A -85,B 0,C 180,E1 -18258.506,E2 -18258.506} C_VEL
LIN {X 0,Y 370.032,Z 285.049,A -85,B 0,C 180,E1 -18260.226,E2 -18260.226} C_VEL
LIN {X 0,Y 373.568,Z 287.359,A -85,B 0,C 180,E1 -18262.024,E2 -18262.024} C_VEL
LIN {X 0,Y 376.284,Z 288.834,A -85,B 0,C 180,E1 -18263.721,E2 -18263.721} C_VEL
LIN {X 0,Y 378.683,Z 289.829,A -85,B 0,C 180,E1 -18265.743,E2 -18265.743} C_VEL
LIN {X 0,Y 379.929,Z 290.267,A -85,B 0,C 180,E1 -18267.3,E2 -18267.3} C_VEL
LIN {X 0,Y 380.613,Z 290.688,A -85,B 0,C 180,E1 -18268.942,E2 -18268.942} C_VEL
LIN {X 0,Y 380.759,Z 290.623,A -85,B 0,C 180,E1 -18270,E2 -18270} C_VEL
LIN {X 0,Y 380.444,Z 290.565,A -85,B 0,C 180,E1 -18271.588,E2 -18271.588} C_VEL
LIN {X 0,Y 379.6,Z 290.062,A -85,B 0,C 180,E1 -18273.184,E2 -18273.184} C_VEL
LIN {X 0,Y 377.821,Z 289.515,A -85,B 0,C 180,E1 -18275.066,E2 -18275.066} C_VEL
LIN {X 0,Y 375.25,Z 288.302,A -85,B 0,C 180,E1 -18276.967,E2 -18276.967} C_VEL
LIN {X 0,Y 371.737,Z 286.24,A -85,B 0,C 180,E1 -18278.954,E2 -18278.954} C_VEL
LIN {X 0,Y 367.919,Z 283.441,A -85,B 0,C 180,E1 -18280.709,E2 -18280.709} C_VEL
LIN {X 0,Y 364.633,Z 280.872,A -85,B 0,C 180,E1 -18282.014,E2 -18282.014} C_VEL
LIN {X 0,Y 359.519,Z 277.859,A -85,B 0,C 180,E1 -18283.755,E2 -18283.755} C_VEL
LIN {X 0,Y 353.674,Z 273.563,A -85,B 0,C 180,E1 -18285.504,E2 -18285.504} C_VEL
LIN {X 0,Y 348.556,Z 269.777,A -85,B 0,C 180,E1 -18286.881,E2 -18286.881} C_VEL
LIN {X 0,Y 342.252,Z 265.019,A -85,B 0,C 180,E1 -18288.423,E2 -18288.423} C_VEL
LIN {X 0,Y 337.005,Z 260.867,A -85,B 0,C 180,E1 -18289.607,E2 -18289.607} C_VEL
LIN {X 0,Y 329.699,Z 254.835,A -85,B 0,C 180,E1 -18291.12,E2 -18291.12} C_VEL
LIN {X 0,Y 321.395,Z 247.841,A -85,B 0,C 180,E1 -18292.659,E2 -18292.659} C_VEL
LIN {X 0,Y 312.666,Z 239.965,A -85,B 0,C 180,E1 -18294.06,E2 -18294.06} C_VEL
LIN {X 0,Y 304.433,Z 232.32,A -85,B 0,C 180,E1 -18295.193,E2 -18295.193} C_VEL
LIN {X 0,Y 292.125,Z 219.704,A -85,B 0,C 180,E1 -18296.721,E2 -18296.721} C_VEL
LIN {X 0,Y 284.054,Z 209.885,A -85,B 0,C 180,E1 -18297.826,E2 -18297.826} C_VEL
LIN {X 0,Y 276.682,Z 199.002,A -85,B 0,C 180,E1 -18298.958,E2 -18298.958} C_VEL
LIN {X 0,Y 264.62,Z 176.751,A -85,B 0,C 180,E1 -18301.115,E2 -18301.115} C_VEL
LIN {X 0,Y 263.301,Z 174.046,A -85,B 0,C 180,E1 -18301.428,E2 -18301.428} C_VEL
LIN {X 0,Y 263.127,Z 173.264,A -85,B 0,C 180,E1 -18301.787,E2 -18301.787} C_VEL
LIN {X 0,Y 263.169,Z 173.166,A -85,B 0,C 180,E1 -18304.122,E2 -18304.122} C_VEL
LIN {X 0,Y 263.162,Z 173.207,A -85,B 0,C 180,E1 -18307.896,E2 -18307.896} C_VEL
LIN {X 0,Y 263.12,Z 173.149,A -85,B 0,C 180,E1 -18311.894,E2 -18311.894} C_VEL
LIN {X 0,Y 263.125,Z 173.208,A -85,B 0,C 180,E1 -18316.15,E2 -18316.15} C_VEL
LIN {X 0,Y 263.11,Z 173.194,A -85,B 0,C 180,E1 -18320.13,E2 -18320.13} C_VEL
LIN {X 0,Y 263.183,Z 173.187,A -85,B 0,C 180,E1 -18324.022,E2 -18324.022} C_VEL
LIN {X 0,Y 263.13,Z 173.205,A -85,B 0,C 180,E1 -18327.712,E2 -18327.712} C_VEL
LIN {X 0,Y 263.197,Z 173.174,A -85,B 0,C 180,E1 -18331.784,E2 -18331.784} C_VEL
LIN {X 0,Y 263.223,Z 173.191,A -85,B 0,C 180,E1 -18335.201,E2 -18335.201} C_VEL
LIN {X 0,Y 263.26,Z 173.161,A -85,B 0,C 180,E1 -18339.694,E2 -18339.694} C_VEL
LIN {X 0,Y 263.348,Z 173.18,A -85,B 0,C 180,E1 -18344.523,E2 -18344.523} C_VEL
LIN {X 0,Y 263.371,Z 173.141,A -85,B 0,C 180,E1 -18349.235,E2 -18349.235} C_VEL
LIN {X 0,Y 263.571,Z 173.132,A -85,B 0,C 180,E1 -18352.339,E2 -18352.339} C_VEL
LIN {X 0,Y 263.749,Z 173.097,A -85,B 0,C 180,E1 -18358.474,E2 -18358.474} C_VEL
LIN {X 0,Y 263.748,Z 173.102,A -85,B 0,C 180,E1 -18361.528,E2 -18361.528} C_VEL
LIN {X 0,Y 263.557,Z 173.132,A -85,B 0,C 180,E1 -18367.663,E2 -18367.663} C_VEL
LIN {X 0,Y 263.354,Z 173.144,A -85,B 0,C 180,E1 -18370.767,E2 -18370.767} C_VEL
LIN {X 0,Y 263.35,Z 173.173,A -85,B 0,C 180,E1 -18375.479,E2 -18375.479} C_VEL
LIN {X 0,Y 263.263,Z 173.165,A -85,B 0,C 180,E1 -18380.307,E2 -18380.307} C_VEL
LIN {X 0,Y 263.208,Z 173.18,A -85,B 0,C 180,E1 -18385.292,E2 -18385.292} C_VEL
LIN {X 0,Y 263.175,Z 173.187,A -85,B 0,C 180,E1 -18388.731,E2 -18388.731} C_VEL
LIN {X 0,Y 263.112,Z 173.193,A -85,B 0,C 180,E1 -18392.738,E2 -18392.738} C_VEL
LIN {X 0,Y 263.193,Z 173.199,A -85,B 0,C 180,E1 -18396.767,E2 -18396.767} C_VEL
LIN {X 0,Y 263.113,Z 173.196,A -85,B 0,C 180,E1 -18399.383,E2 -18399.383} C_VEL
LIN {X 0,Y 262.419,Z 173.283,A -85,B 0,C 180,E1 -18400.66,E2 -18400.66} C_VEL
LIN {X 0,Y 259.551,Z 173.655,A -85,B 0,C 180,E1 -18402.742,E2 -18402.742} C_VEL
LIN {X 0,Y 257.141,Z 173.95,A -85,B 0,C 180,E1 -18404.436,E2 -18404.436} C_VEL
LIN {X 0,Y 256.123,Z 174.076,A -85,B 0,C 180,E1 -18405.749,E2 -18405.749} C_VEL
LIN {X 0,Y 256.047,Z 174.088,A -85,B 0,C 180,E1 -18406.194,E2 -18406.194} C_VEL
LIN {X 0,Y 256.137,Z 174.16,A -85,B 0,C 180,E1 -18410.927,E2 -18410.927} C_VEL
LIN {X 0,Y 257.79,Z 181.566,A -85,B 0,C 180,E1 -18414.874,E2 -18414.874} C_VEL
LIN {X 0,Y 259.02,Z 187.873,A -85,B 0,C 180,E1 -18417.996,E2 -18417.996} C_VEL
LIN {X 0,Y 259.808,Z 190.264,A -85,B 0,C 180,E1 -18418.288,E2 -18418.288} C_VEL
LIN {X 0,Y 265.96,Z 204.022,A -85,B 0,C 180,E1 -18419.52,E2 -18419.52} C_VEL
LIN {X 0,Y 267.572,Z 209.971,A -85,B 0,C 180,E1 -18419.902,E2 -18419.902} C_VEL
LIN {X 0,Y 271.551,Z 230.696,A -85,B 0,C 180,E1 -18420.998,E2 -18420.998} C_VEL
LIN {X 0,Y 272.871,Z 239.587,A -85,B 0,C 180,E1 -18421.412,E2 -18421.412} C_VEL
LIN {X 0,Y 271.094,Z 294.406,A -85,B 0,C 180,E1 -18422.869,E2 -18422.869} C_VEL
LIN {X 0,Y 270.33,Z 304.604,A -85,B 0,C 180,E1 -18423.306,E2 -18423.306} C_VEL
LIN {X 0,Y 269.297,Z 314.072,A -85,B 0,C 180,E1 -18423.871,E2 -18423.871} C_VEL
LIN {X 0,Y 267.984,Z 324.15,A -85,B 0,C 180,E1 -18424.672,E2 -18424.672} C_VEL
LIN {X 0,Y 266.542,Z 333.908,A -85,B 0,C 180,E1 -18425.67,E2 -18425.67} C_VEL
LIN {X 0,Y 264.679,Z 343.97,A -85,B 0,C 180,E1 -18426.943,E2 -18426.943} C_VEL
LIN {X 0,Y 262.331,Z 355.465,A -85,B 0,C 180,E1 -18428.797,E2 -18428.797} C_VEL
LIN {X 0,Y 260.381,Z 364.602,A -85,B 0,C 180,E1 -18430.692,E2 -18430.692} C_VEL
LIN {X 0,Y 259.088,Z 370.98,A -85,B 0,C 180,E1 -18432.283,E2 -18432.283} C_VEL
LIN {X 0,Y 257.636,Z 377.343,A -85,B 0,C 180,E1 -18434.17,E2 -18434.17} C_VEL
LIN {X 0,Y 256.615,Z 381.844,A -85,B 0,C 180,E1 -18435.731,E2 -18435.731} C_VEL
LIN {X 0,Y 255.428,Z 387.336,A -85,B 0,C 180,E1 -18438.091,E2 -18438.091} C_VEL
LIN {X 0,Y 254.643,Z 391.663,A -85,B 0,C 180,E1 -18440.468,E2 -18440.468} C_VEL
LIN {X 0,Y 254.311,Z 394.033,A -85,B 0,C 180,E1 -18442.058,E2 -18442.058} C_VEL
LIN {X 0,Y 253.993,Z 397.018,A -85,B 0,C 180,E1 -18444.961,E2 -18444.961} C_VEL
LIN {X 0,Y 253.954,Z 398.287,A -85,B 0,C 180,E1 -18446.827,E2 -18446.827} C_VEL
LIN {X 0,Y 253.995,Z 398.879,A -85,B 0,C 180,E1 -18448.414,E2 -18448.414} C_VEL
LIN {X 0,Y 254.047,Z 399.035,A -85,B 0,C 180,E1 -18450,E2 -18450} C_VEL
LIN {X 0,Y 253.995,Z 398.879,A -85,B 0,C 180,E1 -18451.586,E2 -18451.586} C_VEL
LIN {X 0,Y 253.951,Z 398.286,A -85,B 0,C 180,E1 -18453.173,E2 -18453.173} C_VEL
LIN {X 0,Y 254.063,Z 395.834,A -85,B 0,C 180,E1 -18456.353,E2 -18456.353} C_VEL
LIN {X 0,Y 254.467,Z 392.882,A -85,B 0,C 180,E1 -18458.737,E2 -18458.737} C_VEL
LIN {X 0,Y 255.116,Z 388.89,A -85,B 0,C 180,E1 -18461.118,E2 -18461.118} C_VEL
LIN {X 0,Y 256.131,Z 383.758,A -85,B 0,C 180,E1 -18463.487,E2 -18463.487} C_VEL
LIN {X 0,Y 257.37,Z 378.498,A -85,B 0,C 180,E1 -18465.441,E2 -18465.441} C_VEL
LIN {X 0,Y 258.78,Z 372.182,A -85,B 0,C 180,E1 -18467.382,E2 -18467.382} C_VEL
LIN {X 0,Y 260.154,Z 365.902,A -85,B 0,C 180,E1 -18468.998,E2 -18468.998} C_VEL
LIN {X 0,Y 261.521,Z 359.303,A -85,B 0,C 180,E1 -18470.448,E2 -18470.448} C_VEL
LIN {X 0,Y 263.233,Z 351.126,A -85,B 0,C 180,E1 -18471.949,E2 -18471.949} C_VEL
LIN {X 0,Y 264.903,Z 342.618,A -85,B 0,C 180,E1 -18473.243,E2 -18473.243} C_VEL
LIN {X 0,Y 266.459,Z 333.906,A -85,B 0,C 180,E1 -18474.338,E2 -18474.338} C_VEL
LIN {X 0,Y 268.007,Z 324.151,A -85,B 0,C 180,E1 -18475.326,E2 -18475.326} C_VEL
LIN {X 0,Y 269.255,Z 314.071,A -85,B 0,C 180,E1 -18476.133,E2 -18476.133} C_VEL
LIN {X 0,Y 270.325,Z 304.632,A -85,B 0,C 180,E1 -18476.693,E2 -18476.693} C_VEL
LIN {X 0,Y 271.091,Z 294.479,A -85,B 0,C 180,E1 -18477.127,E2 -18477.127} C_VEL
LIN {X 0,Y 272.876,Z 239.297,A -85,B 0,C 180,E1 -18478.596,E2 -18478.596} C_VEL
LIN {X 0,Y 269.801,Z 221.134,A -85,B 0,C 180,E1 -18479.492,E2 -18479.492} C_VEL
LIN {X 0,Y 266.348,Z 204.986,A -85,B 0,C 180,E1 -18480.402,E2 -18480.402} C_VEL
LIN {X 0,Y 259.129,Z 188.227,A -85,B 0,C 180,E1 -18481.916,E2 -18481.916} C_VEL
LIN {X 0,Y 258.65,Z 185.872,A -85,B 0,C 180,E1 -18482.917,E2 -18482.917} C_VEL
LIN {X 0,Y 257.023,Z 178.004,A -85,B 0,C 180,E1 -18486.982,E2 -18486.982} C_VEL
LIN {X 0,Y 256.136,Z 174.144,A -85,B 0,C 180,E1 -18489.13,E2 -18489.13} C_VEL
LIN {X 0,Y 256.063,Z 174.091,A -85,B 0,C 180,E1 -18493.326,E2 -18493.326} C_VEL
LIN {X 0,Y 256.071,Z 174.089,A -85,B 0,C 180,E1 -18497.819,E2 -18497.819} C_VEL
LIN {X 0,Y 256.072,Z 174.074,A -85,B 0,C 180,E1 -18500.857,E2 -18500.857} C_VEL
LIN {X 0,Y 256.139,Z 174.08,A -85,B 0,C 180,E1 -18502.868,E2 -18502.868} C_VEL
LIN {X 0,Y 256.068,Z 174.066,A -85,B 0,C 180,E1 -18506.706,E2 -18506.706} C_VEL
LIN {X 0,Y 256.111,Z 174.077,A -85,B 0,C 180,E1 -18510.399,E2 -18510.399} C_VEL
LIN {X 0,Y 256.188,Z 174.055,A -85,B 0,C 180,E1 -18514.861,E2 -18514.861} C_VEL
LIN {X 0,Y 256.166,Z 174.058,A -85,B 0,C 180,E1 -18519.104,E2 -18519.104} C_VEL
LIN {X 0,Y 256.299,Z 174.049,A -85,B 0,C 180,E1 -18524.084,E2 -18524.084} C_VEL
LIN {X 0,Y 256.294,Z 174.049,A -85,B 0,C 180,E1 -18527.327,E2 -18527.327} C_VEL
LIN {X 0,Y 256.514,Z 174.004,A -85,B 0,C 180,E1 -18532.125,E2 -18532.125} C_VEL
LIN {X 0,Y 256.496,Z 174.026,A -85,B 0,C 180,E1 -18536.858,E2 -18536.858} C_VEL
LIN {X 0,Y 256.755,Z 173.958,A -85,B 0,C 180,E1 -18539.999,E2 -18539.999} C_VEL
LIN {X 0,Y 256.497,Z 174.023,A -85,B 0,C 180,E1 -18543.141,E2 -18543.141} C_VEL
LIN {X 0,Y 256.538,Z 174.005,A -85,B 0,C 180,E1 -18547.872,E2 -18547.872} C_VEL
LIN {X 0,Y 256.307,Z 174.023,A -85,B 0,C 180,E1 -18551.065,E2 -18551.065} C_VEL
LIN {X 0,Y 256.297,Z 174.053,A -85,B 0,C 180,E1 -18555.914,E2 -18555.914} C_VEL
LIN {X 0,Y 256.163,Z 174.053,A -85,B 0,C 180,E1 -18560.894,E2 -18560.894} C_VEL
LIN {X 0,Y 256.185,Z 174.061,A -85,B 0,C 180,E1 -18565.138,E2 -18565.138} C_VEL
LIN {X 0,Y 256.11,Z 174.074,A -85,B 0,C 180,E1 -18569.599,E2 -18569.599} C_VEL
LIN {X 0,Y 256.081,Z 174.067,A -85,B 0,C 180,E1 -18573.29,E2 -18573.29} C_VEL
LIN {X 0,Y 256.125,Z 174.082,A -85,B 0,C 180,E1 -18577.274,E2 -18577.274} C_VEL
LIN {X 0,Y 256.052,Z 174.072,A -85,B 0,C 180,E1 -18581.203,E2 -18581.203} C_VEL
LIN {X 0,Y 256.058,Z 174.055,A -85,B 0,C 180,E1 -18585.529,E2 -18585.529} C_VEL
LIN {X 0,Y 256.052,Z 174.032,A -85,B 0,C 180,E1 -18588.797,E2 -18588.797} C_VEL
LIN {X 0,Y 256.141,Z 174.069,A -85,B 0,C 180,E1 -18592.87,E2 -18592.87} C_VEL
LIN {X 0,Y 256.098,Z 174.11,A -85,B 0,C 180,E1 -18597.302,E2 -18597.302} C_VEL
LIN {X 0,Y 256.254,Z 174.957,A -85,B 0,C 180,E1 -18597.642,E2 -18597.642} C_VEL
LIN {X 0,Y 257.768,Z 177.866,A -85,B 0,C 180,E1 -18597.991,E2 -18597.991} C_VEL
LIN {X 0,Y 266.202,Z 193.397,A -85,B 0,C 180,E1 -18599.605,E2 -18599.605} C_VEL
LIN {X 0,Y 273.3,Z 206.203,A -85,B 0,C 180,E1 -18600.859,E2 -18600.859} C_VEL
LIN {X 0,Y 281.714,Z 218.059,A -85,B 0,C 180,E1 -18602.152,E2 -18602.152} C_VEL
LIN {X 0,Y 292.369,Z 230.023,A -85,B 0,C 180,E1 -18603.581,E2 -18603.581} C_VEL
LIN {X 0,Y 304.531,Z 241.914,A -85,B 0,C 180,E1 -18605.075,E2 -18605.075} C_VEL
LIN {X 0,Y 314.063,Z 250.348,A -85,B 0,C 180,E1 -18606.405,E2 -18606.405} C_VEL
LIN {X 0,Y 322.682,Z 257.818,A -85,B 0,C 180,E1 -18607.829,E2 -18607.829} C_VEL
LIN {X 0,Y 331.242,Z 264.844,A -85,B 0,C 180,E1 -18609.454,E2 -18609.454} C_VEL
LIN {X 0,Y 339.212,Z 270.922,A -85,B 0,C 180,E1 -18611.147,E2 -18611.147} C_VEL
LIN {X 0,Y 346.111,Z 276.148,A -85,B 0,C 180,E1 -18612.78,E2 -18612.78} C_VEL
LIN {X 0,Y 351.335,Z 279.928,A -85,B 0,C 180,E1 -18614.145,E2 -18614.145} C_VEL
LIN {X 0,Y 356.389,Z 283.661,A -85,B 0,C 180,E1 -18615.608,E2 -18615.608} C_VEL
LIN {X 0,Y 361.381,Z 286.766,A -85,B 0,C 180,E1 -18617.183,E2 -18617.183} C_VEL
LIN {X 0,Y 364.571,Z 288.717,A -85,B 0,C 180,E1 -18618.33,E2 -18618.33} C_VEL
LIN {X 0,Y 368.887,Z 292.056,A -85,B 0,C 180,E1 -18620.127,E2 -18620.127} C_VEL
LIN {X 0,Y 372.366,Z 294.276,A -85,B 0,C 180,E1 -18621.851,E2 -18621.851} C_VEL
LIN {X 0,Y 375.376,Z 295.884,A -85,B 0,C 180,E1 -18623.706,E2 -18623.706} C_VEL
LIN {X 0,Y 377.8,Z 296.852,A -85,B 0,C 180,E1 -18625.733,E2 -18625.733} C_VEL
LIN {X 0,Y 379.058,Z 297.315,A -85,B 0,C 180,E1 -18627.294,E2 -18627.294} C_VEL
LIN {X 0,Y 379.744,Z 297.734,A -85,B 0,C 180,E1 -18628.94,E2 -18628.94} C_VEL
LIN {X 0,Y 379.893,Z 297.67,A -85,B 0,C 180,E1 -18630,E2 -18630} C_VEL
LIN {X 0,Y 379.625,Z 297.631,A -85,B 0,C 180,E1 -18631.43,E2 -18631.43} C_VEL
LIN {X 0,Y 378.723,Z 297.103,A -85,B 0,C 180,E1 -18633.191,E2 -18633.191} C_VEL
LIN {X 0,Y 376.929,Z 296.561,A -85,B 0,C 180,E1 -18635.078,E2 -18635.078} C_VEL
LIN {X 0,Y 374.246,Z 295.287,A -85,B 0,C 180,E1 -18637.04,E2 -18637.04} C_VEL
LIN {X 0,Y 370.773,Z 293.323,A -85,B 0,C 180,E1 -18638.978,E2 -18638.978} C_VEL
LIN {X 0,Y 367.027,Z 290.665,A -85,B 0,C 180,E1 -18640.686,E2 -18640.686} C_VEL
LIN {X 0,Y 363.238,Z 287.738,A -85,B 0,C 180,E1 -18642.174,E2 -18642.174} C_VEL
LIN {X 0,Y 358.36,Z 284.952,A -85,B 0,C 180,E1 -18643.8,E2 -18643.8} C_VEL
LIN {X 0,Y 352.643,Z 280.97,A -85,B 0,C 180,E1 -18645.489,E2 -18645.489} C_VEL
LIN {X 0,Y 347.921,Z 277.359,A -85,B 0,C 180,E1 -18646.763,E2 -18646.763} C_VEL
LIN {X 0,Y 341.435,Z 272.768,A -85,B 0,C 180,E1 -18648.339,E2 -18648.339} C_VEL
LIN {X 0,Y 334.592,Z 267.364,A -85,B 0,C 180,E1 -18649.859,E2 -18649.859} C_VEL
LIN {X 0,Y 327.346,Z 261.569,A -85,B 0,C 180,E1 -18651.317,E2 -18651.317} C_VEL
LIN {X 0,Y 319.005,Z 254.741,A -85,B 0,C 180,E1 -18652.799,E2 -18652.799} C_VEL
LIN {X 0,Y 311.603,Z 248.267,A -85,B 0,C 180,E1 -18653.956,E2 -18653.956} C_VEL
LIN {X 0,Y 302.429,Z 239.993,A -85,B 0,C 180,E1 -18655.194,E2 -18655.194} C_VEL
LIN {X 0,Y 288.672,Z 226.129,A -85,B 0,C 180,E1 -18656.894,E2 -18656.894} C_VEL
LIN {X 0,Y 279.566,Z 215.22,A -85,B 0,C 180,E1 -18658.164,E2 -18658.164} C_VEL
LIN {X 0,Y 271.753,Z 203.727,A -85,B 0,C 180,E1 -18659.398,E2 -18659.398} C_VEL
LIN {X 0,Y 259.577,Z 181.122,A -85,B 0,C 180,E1 -18661.654,E2 -18661.654} C_VEL
LIN {X 0,Y 256.314,Z 175.117,A -85,B 0,C 180,E1 -18662.335,E2 -18662.335} C_VEL
LIN {X 0,Y 256.098,Z 174.151,A -85,B 0,C 180,E1 -18662.699,E2 -18662.699} C_VEL
LIN {X 0,Y 256.116,Z 174.044,A -85,B 0,C 180,E1 -18665.187,E2 -18665.187} C_VEL
LIN {X 0,Y 256.083,Z 174.066,A -85,B 0,C 180,E1 -18669.139,E2 -18669.139} C_VEL
LIN {X 0,Y 256.06,Z 174.035,A -85,B 0,C 180,E1 -18673.327,E2 -18673.327} C_VEL
LIN {X 0,Y 256.069,Z 174.079,A -85,B 0,C 180,E1 -18677.819,E2 -18677.819} C_VEL
LIN {X 0,Y 256.084,Z 174.077,A -85,B 0,C 180,E1 -18680.861,E2 -18680.861} C_VEL
LIN {X 0,Y 256.117,Z 174.058,A -85,B 0,C 180,E1 -18684.814,E2 -18684.814} C_VEL
LIN {X 0,Y 256.089,Z 174.087,A -85,B 0,C 180,E1 -18688.573,E2 -18688.573} C_VEL
LIN {X 0,Y 256.138,Z 174.049,A -85,B 0,C 180,E1 -18692.197,E2 -18692.197} C_VEL
LIN {X 0,Y 256.164,Z 174.073,A -85,B 0,C 180,E1 -18695.7,E2 -18695.7} C_VEL
LIN {X 0,Y 256.163,Z 174.053,A -85,B 0,C 180,E1 -18699.106,E2 -18699.106} C_VEL
LIN {X 0,Y 256.297,Z 174.053,A -85,B 0,C 180,E1 -18704.086,E2 -18704.086} C_VEL
LIN {X 0,Y 256.307,Z 174.023,A -85,B 0,C 180,E1 -18708.935,E2 -18708.935} C_VEL
LIN {X 0,Y 256.538,Z 174.005,A -85,B 0,C 180,E1 -18712.128,E2 -18712.128} C_VEL
LIN {X 0,Y 256.712,Z 173.973,A -85,B 0,C 180,E1 -18718.432,E2 -18718.432} C_VEL
LIN {X 0,Y 256.711,Z 173.978,A -85,B 0,C 180,E1 -18721.57,E2 -18721.57} C_VEL
LIN {X 0,Y 256.48,Z 174.031,A -85,B 0,C 180,E1 -18726.294,E2 -18726.294} C_VEL
LIN {X 0,Y 256.425,Z 174,A -85,B 0,C 180,E1 -18729.466,E2 -18729.466} C_VEL
LIN {X 0,Y 256.255,Z 174.061,A -85,B 0,C 180,E1 -18734.291,E2 -18734.291} C_VEL
LIN {X 0,Y 256.21,Z 174.036,A -85,B 0,C 180,E1 -18737.563,E2 -18737.563} C_VEL
LIN {X 0,Y 256.157,Z 174.061,A -85,B 0,C 180,E1 -18741.121,E2 -18741.121} C_VEL
LIN {X 0,Y 256.188,Z 174.055,A -85,B 0,C 180,E1 -18745.139,E2 -18745.139} C_VEL
LIN {X 0,Y 256.111,Z 174.077,A -85,B 0,C 180,E1 -18749.601,E2 -18749.601} C_VEL
LIN {X 0,Y 256.068,Z 174.066,A -85,B 0,C 180,E1 -18753.294,E2 -18753.294} C_VEL
LIN {X 0,Y 256.123,Z 174.082,A -85,B 0,C 180,E1 -18757.274,E2 -18757.274} C_VEL
LIN {X 0,Y 256.055,Z 174.078,A -85,B 0,C 180,E1 -18761.204,E2 -18761.204} C_VEL
LIN {X 0,Y 256.055,Z 174.083,A -85,B 0,C 180,E1 -18765.532,E2 -18765.532} C_VEL
LIN {X 0,Y 256.047,Z 174.088,A -85,B 0,C 180,E1 -18766.194,E2 -18766.194} C_VEL
LIN {X 0,Y 255.345,Z 174.19,A -85,B 0,C 180,E1 -18767.087,E2 -18767.087} C_VEL
LIN {X 0,Y 252.413,Z 174.516,A -85,B 0,C 180,E1 -18768.488,E2 -18768.488} C_VEL
LIN {X 0,Y 249.692,Z 174.992,A -85,B 0,C 180,E1 -18769.889,E2 -18769.889} C_VEL
LIN {X 0,Y 249.247,Z 175.772,A -85,B 0,C 180,E1 -18770.613,E2 -18770.613} C_VEL
LIN {X 0,Y 249.286,Z 176.002,A -85,B 0,C 180,E1 -18770.754,E2 -18770.754} C_VEL
LIN {X 0,Y 250.781,Z 182.57,A -85,B 0,C 180,E1 -18774.363,E2 -18774.363} C_VEL
LIN {X 0,Y 251.815,Z 187.703,A -85,B 0,C 180,E1 -18776.98,E2 -18776.98} C_VEL
LIN {X 0,Y 253.265,Z 191.308,A -85,B 0,C 180,E1 -18777.41,E2 -18777.41} C_VEL
LIN {X 0,Y 260.641,Z 208.05,A -85,B 0,C 180,E1 -18778.961,E2 -18778.961} C_VEL
LIN {X 0,Y 264.63,Z 227.746,A -85,B 0,C 180,E1 -18780.081,E2 -18780.081} C_VEL
LIN {X 0,Y 266.614,Z 240.681,A -85,B 0,C 180,E1 -18780.715,E2 -18780.715} C_VEL
LIN {X 0,Y 264.849,Z 293.576,A -85,B 0,C 180,E1 -18782.147,E2 -18782.147} C_VEL
LIN {X 0,Y 264.084,Z 303.753,A -85,B 0,C 180,E1 -18782.582,E2 -18782.582} C_VEL
LIN {X 0,Y 262.931,Z 313.88,A -85,B 0,C 180,E1 -18783.189,E2 -18783.189} C_VEL
LIN {X 0,Y 261.591,Z 323.959,A -85,B 0,C 180,E1 -18784.008,E2 -18784.008} C_VEL
LIN {X 0,Y 260.089,Z 333.716,A -85,B 0,C 180,E1 -18785.026,E2 -18785.026} C_VEL
LIN {X 0,Y 258.13,Z 343.777,A -85,B 0,C 180,E1 -18786.323,E2 -18786.323} C_VEL
LIN {X 0,Y 255.708,Z 355.273,A -85,B 0,C 180,E1 -18788.22,E2 -18788.22} C_VEL
LIN {X 0,Y 253.675,Z 364.41,A -85,B 0,C 180,E1 -18790.161,E2 -18790.161} C_VEL
LIN {X 0,Y 252.268,Z 370.929,A -85,B 0,C 180,E1 -18791.831,E2 -18791.831} C_VEL
LIN {X 0,Y 250.772,Z 377.15,A -85,B 0,C 180,E1 -18793.725,E2 -18793.725} C_VEL
LIN {X 0,Y 249.704,Z 381.651,A -85,B 0,C 180,E1 -18795.327,E2 -18795.327} C_VEL
LIN {X 0,Y 248.435,Z 387.143,A -85,B 0,C 180,E1 -18797.751,E2 -18797.751} C_VEL
LIN {X 0,Y 247.615,Z 391.471,A -85,B 0,C 180,E1 -18800.195,E2 -18800.195} C_VEL
LIN {X 0,Y 247.263,Z 393.841,A -85,B 0,C 180,E1 -18801.83,E2 -18801.83} C_VEL
LIN {X 0,Y 247.011,Z 395.642,A -85,B 0,C 180,E1 -18803.465,E2 -18803.465} C_VEL
LIN {X 0,Y 246.858,Z 398.095,A -85,B 0,C 180,E1 -18806.736,E2 -18806.736} C_VEL
LIN {X 0,Y 246.905,Z 398.687,A -85,B 0,C 180,E1 -18808.369,E2 -18808.369} C_VEL
LIN {X 0,Y 246.976,Z 398.844,A -85,B 0,C 180,E1 -18810,E2 -18810} C_VEL
LIN {X 0,Y 246.904,Z 398.687,A -85,B 0,C 180,E1 -18811.631,E2 -18811.631} C_VEL
LIN {X 0,Y 246.855,Z 398.095,A -85,B 0,C 180,E1 -18813.264,E2 -18813.264} C_VEL
LIN {X 0,Y 246.985,Z 395.642,A -85,B 0,C 180,E1 -18816.536,E2 -18816.536} C_VEL
LIN {X 0,Y 247.412,Z 392.689,A -85,B 0,C 180,E1 -18818.988,E2 -18818.988} C_VEL
LIN {X 0,Y 248.128,Z 388.698,A -85,B 0,C 180,E1 -18821.436,E2 -18821.436} C_VEL
LIN {X 0,Y 249.201,Z 383.566,A -85,B 0,C 180,E1 -18823.87,E2 -18823.87} C_VEL
LIN {X 0,Y 250.512,Z 378.306,A -85,B 0,C 180,E1 -18825.874,E2 -18825.874} C_VEL
LIN {X 0,Y 252.009,Z 371.99,A -85,B 0,C 180,E1 -18827.864,E2 -18827.864} C_VEL
LIN {X 0,Y 253.709,Z 364.411,A -85,B 0,C 180,E1 -18829.836,E2 -18829.836} C_VEL
LIN {X 0,Y 255.72,Z 355.273,A -85,B 0,C 180,E1 -18831.778,E2 -18831.778} C_VEL
LIN {X 0,Y 258.126,Z 343.777,A -85,B 0,C 180,E1 -18833.678,E2 -18833.678} C_VEL
LIN {X 0,Y 260.018,Z 333.714,A -85,B 0,C 180,E1 -18834.981,E2 -18834.981} C_VEL
LIN {X 0,Y 261.612,Z 323.96,A -85,B 0,C 180,E1 -18835.99,E2 -18835.99} C_VEL
LIN {X 0,Y 262.912,Z 313.879,A -85,B 0,C 180,E1 -18836.813,E2 -18836.813} C_VEL
LIN {X 0,Y 264.086,Z 303.786,A -85,B 0,C 180,E1 -18837.416,E2 -18837.416} C_VEL
LIN {X 0,Y 264.848,Z 293.612,A -85,B 0,C 180,E1 -18837.849,E2 -18837.849} C_VEL
LIN {X 0,Y 266.596,Z 240.003,A -85,B 0,C 180,E1 -18839.308,E2 -18839.308} C_VEL
LIN {X 0,Y 263.692,Z 222.76,A -85,B 0,C 180,E1 -18840.189,E2 -18840.189} C_VEL
LIN {X 0,Y 260.515,Z 207.744,A -85,B 0,C 180,E1 -18841.065,E2 -18841.065} C_VEL
LIN {X 0,Y 253.503,Z 191.652,A -85,B 0,C 180,E1 -18842.544,E2 -18842.544} C_VEL
LIN {X 0,Y 251.852,Z 187.908,A -85,B 0,C 180,E1 -18842.968,E2 -18842.968} C_VEL
LIN {X 0,Y 250.762,Z 182.588,A -85,B 0,C 180,E1 -18845.631,E2 -18845.631} C_VEL
LIN {X 0,Y 249.223,Z 175.763,A -85,B 0,C 180,E1 -18849.382,E2 -18849.382} C_VEL
LIN {X 0,Y 249.012,Z 174.941,A -85,B 0,C 180,E1 -18850.084,E2 -18850.084} C_VEL
LIN {X 0,Y 249.01,Z 174.962,A -85,B 0,C 180,E1 -18852.792,E2 -18852.792} C_VEL
LIN {X 0,Y 249.01,Z 174.97,A -85,B 0,C 180,E1 -18857.361,E2 -18857.361} C_VEL
LIN {X 0,Y 249.029,Z 174.959,A -85,B 0,C 180,E1 -18861.619,E2 -18861.619} C_VEL
LIN {X 0,Y 249.046,Z 174.937,A -85,B 0,C 180,E1 -18865.639,E2 -18865.639} C_VEL
LIN {X 0,Y 249.051,Z 174.962,A -85,B 0,C 180,E1 -18869.472,E2 -18869.472} C_VEL
LIN {X 0,Y 249.072,Z 174.926,A -85,B 0,C 180,E1 -18873.161,E2 -18873.161} C_VEL
LIN {X 0,Y 249.079,Z 174.956,A -85,B 0,C 180,E1 -18876.732,E2 -18876.732} C_VEL
LIN {X 0,Y 249.109,Z 174.919,A -85,B 0,C 180,E1 -18880.211,E2 -18880.211} C_VEL
LIN {X 0,Y 249.242,Z 174.919,A -85,B 0,C 180,E1 -18883.621,E2 -18883.621} C_VEL
LIN {X 0,Y 249.243,Z 174.907,A -85,B 0,C 180,E1 -18888.615,E2 -18888.615} C_VEL
LIN {X 0,Y 249.453,Z 174.878,A -85,B 0,C 180,E1 -18891.901,E2 -18891.901} C_VEL
LIN {X 0,Y 249.295,Z 174.932,A -85,B 0,C 180,E1 -18895.148,E2 -18895.148} C_VEL
LIN {X 0,Y 249.673,Z 174.854,A -85,B 0,C 180,E1 -18898.386,E2 -18898.386} C_VEL
LIN {X 0,Y 249.674,Z 174.849,A -85,B 0,C 180,E1 -18901.612,E2 -18901.612} C_VEL
LIN {X 0,Y 249.449,Z 174.9,A -85,B 0,C 180,E1 -18906.73,E2 -18906.73} C_VEL
LIN {X 0,Y 249.386,Z 174.877,A -85,B 0,C 180,E1 -18909.734,E2 -18909.734} C_VEL
LIN {X 0,Y 249.203,Z 174.943,A -85,B 0,C 180,E1 -18914.703,E2 -18914.703} C_VEL
LIN {X 0,Y 249.136,Z 174.916,A -85,B 0,C 180,E1 -18918.077,E2 -18918.077} C_VEL
LIN {X 0,Y 249.084,Z 174.946,A -85,B 0,C 180,E1 -18921.517,E2 -18921.517} C_VEL
LIN {X 0,Y 249.127,Z 174.935,A -85,B 0,C 180,E1 -18925.481,E2 -18925.481} C_VEL
LIN {X 0,Y 249.08,Z 174.94,A -85,B 0,C 180,E1 -18928.993,E2 -18928.993} C_VEL
LIN {X 0,Y 249.032,Z 174.958,A -85,B 0,C 180,E1 -18932.424,E2 -18932.424} C_VEL
LIN {X 0,Y 249.065,Z 174.95,A -85,B 0,C 180,E1 -18936.338,E2 -18936.338} C_VEL
LIN {X 0,Y 249.022,Z 174.946,A -85,B 0,C 180,E1 -18940.474,E2 -18940.474} C_VEL
LIN {X 0,Y 249.003,Z 174.949,A -85,B 0,C 180,E1 -18944.878,E2 -18944.878} C_VEL
LIN {X 0,Y 249.014,Z 174.905,A -85,B 0,C 180,E1 -18947.363,E2 -18947.363} C_VEL
LIN {X 0,Y 249.034,Z 174.963,A -85,B 0,C 180,E1 -18951.621,E2 -18951.621} C_VEL
LIN {X 0,Y 249.057,Z 174.921,A -85,B 0,C 180,E1 -18955.642,E2 -18955.642} C_VEL
LIN {X 0,Y 249.09,Z 175.184,A -85,B 0,C 180,E1 -18956.447,E2 -18956.447} C_VEL
LIN {X 0,Y 249.428,Z 176.529,A -85,B 0,C 180,E1 -18956.719,E2 -18956.719} C_VEL
LIN {X 0,Y 258.323,Z 192.371,A -85,B 0,C 180,E1 -18958.533,E2 -18958.533} C_VEL
LIN {X 0,Y 267.232,Z 209.02,A -85,B 0,C 180,E1 -18960.211,E2 -18960.211} C_VEL
LIN {X 0,Y 275.73,Z 221.429,A -85,B 0,C 180,E1 -18961.586,E2 -18961.586} C_VEL
LIN {X 0,Y 286.256,Z 233.541,A -85,B 0,C 180,E1 -18963.063,E2 -18963.063} C_VEL
LIN {X 0,Y 299.664,Z 246.858,A -85,B 0,C 180,E1 -18964.721,E2 -18964.721} C_VEL
LIN {X 0,Y 308.982,Z 255.078,A -85,B 0,C 180,E1 -18965.924,E2 -18965.924} C_VEL
LIN {X 0,Y 317.117,Z 261.998,A -85,B 0,C 180,E1 -18967.15,E2 -18967.15} C_VEL
LIN {X 0,Y 324.018,Z 267.496,A -85,B 0,C 180,E1 -18968.329,E2 -18968.329} C_VEL
LIN {X 0,Y 330.504,Z 272.699,A -85,B 0,C 180,E1 -18969.562,E2 -18969.562} C_VEL
LIN {X 0,Y 337.465,Z 277.978,A -85,B 0,C 180,E1 -18971.024,E2 -18971.024} C_VEL
LIN {X 0,Y 344.956,Z 283.403,A -85,B 0,C 180,E1 -18972.767,E2 -18972.767} C_VEL
LIN {X 0,Y 351.434,Z 288.181,A -85,B 0,C 180,E1 -18974.475,E2 -18974.475} C_VEL
LIN {X 0,Y 356.695,Z 291.734,A -85,B 0,C 180,E1 -18976.011,E2 -18976.011} C_VEL
LIN {X 0,Y 361.547,Z 294.504,A -85,B 0,C 180,E1 -18977.579,E2 -18977.579} C_VEL
LIN {X 0,Y 366.407,Z 298.149,A -85,B 0,C 180,E1 -18979.462,E2 -18979.462} C_VEL
LIN {X 0,Y 370.265,Z 300.703,A -85,B 0,C 180,E1 -18981.266,E2 -18981.266} C_VEL
LIN {X 0,Y 373.74,Z 302.597,A -85,B 0,C 180,E1 -18983.263,E2 -18983.263} C_VEL
LIN {X 0,Y 376.271,Z 303.731,A -85,B 0,C 180,E1 -18985.186,E2 -18985.186} C_VEL
LIN {X 0,Y 377.956,Z 304.267,A -85,B 0,C 180,E1 -18987.069,E2 -18987.069} C_VEL
LIN {X 0,Y 378.777,Z 304.767,A -85,B 0,C 180,E1 -18988.937,E2 -18988.937} C_VEL
LIN {X 0,Y 378.931,Z 304.687,A -85,B 0,C 180,E1 -18990,E2 -18990} C_VEL
LIN {X 0,Y 378.671,Z 304.666,A -85,B 0,C 180,E1 -18991.434,E2 -18991.434} C_VEL
LIN {X 0,Y 377.771,Z 304.121,A -85,B 0,C 180,E1 -18993.199,E2 -18993.199} C_VEL
LIN {X 0,Y 375.953,Z 303.595,A -85,B 0,C 180,E1 -18995.091,E2 -18995.091} C_VEL
LIN {X 0,Y 373.249,Z 302.341,A -85,B 0,C 180,E1 -18997.059,E2 -18997.059} C_VEL
LIN {X 0,Y 369.921,Z 300.473,A -85,B 0,C 180,E1 -18998.916,E2 -18998.916} C_VEL
LIN {X 0,Y 365.983,Z 297.819,A -85,B 0,C 180,E1 -19000.716,E2 -19000.716} C_VEL
LIN {X 0,Y 361.439,Z 294.451,A -85,B 0,C 180,E1 -19002.458,E2 -19002.458} C_VEL
LIN {X 0,Y 356.567,Z 291.678,A -85,B 0,C 180,E1 -19004.027,E2 -19004.027} C_VEL
LIN {X 0,Y 351.255,Z 288.044,A -85,B 0,C 180,E1 -19005.575,E2 -19005.575} C_VEL
LIN {X 0,Y 344.808,Z 283.282,A -85,B 0,C 180,E1 -19007.272,E2 -19007.272} C_VEL
LIN {X 0,Y 337.48,Z 278.018,A -85,B 0,C 180,E1 -19008.972,E2 -19008.972} C_VEL
LIN {X 0,Y 330.154,Z 272.395,A -85,B 0,C 180,E1 -19010.509,E2 -19010.509} C_VEL
LIN {X 0,Y 323.467,Z 267.053,A -85,B 0,C 180,E1 -19011.765,E2 -19011.765} C_VEL
LIN {X 0,Y 316.938,Z 261.881,A -85,B 0,C 180,E1 -19012.878,E2 -19012.878} C_VEL
LIN {X 0,Y 308.679,Z 254.796,A -85,B 0,C 180,E1 -19014.121,E2 -19014.121} C_VEL
LIN {X 0,Y 298.549,Z 245.856,A -85,B 0,C 180,E1 -19015.412,E2 -19015.412} C_VEL
LIN {X 0,Y 284.411,Z 231.611,A -85,B 0,C 180,E1 -19017.181,E2 -19017.181} C_VEL
LIN {X 0,Y 275.217,Z 220.685,A -85,B 0,C 180,E1 -19018.494,E2 -19018.494} C_VEL
LIN {X 0,Y 266.932,Z 208.568,A -85,B 0,C 180,E1 -19019.84,E2 -19019.84} C_VEL
LIN {X 0,Y 257.917,Z 191.558,A -85,B 0,C 180,E1 -19021.549,E2 -19021.549} C_VEL
LIN {X 0,Y 250.463,Z 178.382,A -85,B 0,C 180,E1 -19023.051,E2 -19023.051} C_VEL
LIN {X 0,Y 249.202,Z 175.7,A -85,B 0,C 180,E1 -19023.399,E2 -19023.399} C_VEL
LIN {X 0,Y 249.044,Z 174.988,A -85,B 0,C 180,E1 -19023.777,E2 -19023.777} C_VEL
LIN {X 0,Y 249.052,Z 174.965,A -85,B 0,C 180,E1 -19027.804,E2 -19027.804} C_VEL
LIN {X 0,Y 249.021,Z 174.915,A -85,B 0,C 180,E1 -19030.475,E2 -19030.475} C_VEL
LIN {X 0,Y 249.003,Z 174.942,A -85,B 0,C 180,E1 -19034.879,E2 -19034.879} C_VEL
LIN {X 0,Y 249.014,Z 174.965,A -85,B 0,C 180,E1 -19037.364,E2 -19037.364} C_VEL
LIN {X 0,Y 249.034,Z 174.965,A -85,B 0,C 180,E1 -19041.622,E2 -19041.622} C_VEL
LIN {X 0,Y 249.057,Z 174.935,A -85,B 0,C 180,E1 -19045.643,E2 -19045.643} C_VEL
LIN {X 0,Y 249.048,Z 174.963,A -85,B 0,C 180,E1 -19049.474,E2 -19049.474} C_VEL
LIN {X 0,Y 249.07,Z 174.929,A -85,B 0,C 180,E1 -19053.163,E2 -19053.163} C_VEL
LIN {X 0,Y 249.076,Z 174.959,A -85,B 0,C 180,E1 -19056.733,E2 -19056.733} C_VEL
LIN {X 0,Y 249.107,Z 174.918,A -85,B 0,C 180,E1 -19060.212,E2 -19060.212} C_VEL
LIN {X 0,Y 249.239,Z 174.929,A -85,B 0,C 180,E1 -19063.623,E2 -19063.623} C_VEL
LIN {X 0,Y 249.25,Z 174.905,A -85,B 0,C 180,E1 -19068.617,E2 -19068.617} C_VEL
LIN {X 0,Y 249.479,Z 174.88,A -85,B 0,C 180,E1 -19071.904,E2 -19071.904} C_VEL
LIN {X 0,Y 249.434,Z 174.903,A -85,B 0,C 180,E1 -19076.77,E2 -19076.77} C_VEL
LIN {X 0,Y 249.719,Z 174.834,A -85,B 0,C 180,E1 -19080.001,E2 -19080.001} C_VEL
LIN {X 0,Y 249.433,Z 174.907,A -85,B 0,C 180,E1 -19083.231,E2 -19083.231} C_VEL
LIN {X 0,Y 249.452,Z 174.903,A -85,B 0,C 180,E1 -19086.472,E2 -19086.472} C_VEL
LIN {X 0,Y 249.342,Z 174.881,A -85,B 0,C 180,E1 -19089.737,E2 -19089.737} C_VEL
LIN {X 0,Y 249.205,Z 174.94,A -85,B 0,C 180,E1 -19094.704,E2 -19094.704} C_VEL
LIN {X 0,Y 249.138,Z 174.912,A -85,B 0,C 180,E1 -19098.078,E2 -19098.078} C_VEL
LIN {X 0,Y 249.087,Z 174.946,A -85,B 0,C 180,E1 -19101.519,E2 -19101.519} C_VEL
LIN {X 0,Y 249.13,Z 174.929,A -85,B 0,C 180,E1 -19105.483,E2 -19105.483} C_VEL
LIN {X 0,Y 249.08,Z 174.944,A -85,B 0,C 180,E1 -19108.993,E2 -19108.993} C_VEL
LIN {X 0,Y 249.031,Z 174.951,A -85,B 0,C 180,E1 -19112.427,E2 -19112.427} C_VEL
LIN {X 0,Y 249.055,Z 174.956,A -85,B 0,C 180,E1 -19116.342,E2 -19116.342} C_VEL
LIN {X 0,Y 249.007,Z 174.95,A -85,B 0,C 180,E1 -19120.479,E2 -19120.479} C_VEL
LIN {X 0,Y 248.994,Z 174.958,A -85,B 0,C 180,E1 -19124.882,E2 -19124.882} C_VEL
LIN {X 0,Y 249.017,Z 174.958,A -85,B 0,C 180,E1 -19127.364,E2 -19127.364} C_VEL
LIN {X 0,Y 249.05,Z 175.066,A -85,B 0,C 180,E1 -19130.192,E2 -19130.192} C_VEL
LIN {X 0,Y 249.286,Z 176.002,A -85,B 0,C 180,E1 -19130.754,E2 -19130.754} C_VEL
LIN {X 0,Y 249.012,Z 177.674,A -85,B 0,C 180,E1 -19131.577,E2 -19131.577} C_VEL
LIN {X 0,Y 246.808,Z 180.823,A -85,B 0,C 180,E1 -19132.853,E2 -19132.853} C_VEL
LIN {X 0,Y 244.524,Z 183.984,A -85,B 0,C 180,E1 -19134.15,E2 -19134.15} C_VEL
LIN {X 0,Y 244.164,Z 185.696,A -85,B 0,C 180,E1 -19134.995,E2 -19134.995} C_VEL
LIN {X 0,Y 244.581,Z 187.716,A -85,B 0,C 180,E1 -19135.925,E2 -19135.925} C_VEL
LIN {X 0,Y 249.5,Z 198.463,A -85,B 0,C 180,E1 -19137.1,E2 -19137.1} C_VEL
LIN {X 0,Y 254.969,Z 211.134,A -85,B 0,C 180,E1 -19138.297,E2 -19138.297} C_VEL
LIN {X 0,Y 259.104,Z 232.569,A -85,B 0,C 180,E1 -19139.532,E2 -19139.532} C_VEL
LIN {X 0,Y 260.407,Z 241.8,A -85,B 0,C 180,E1 -19139.987,E2 -19139.987} C_VEL
LIN {X 0,Y 258.573,Z 294.016,A -85,B 0,C 180,E1 -19141.437,E2 -19141.437} C_VEL
LIN {X 0,Y 257.705,Z 304.606,A -85,B 0,C 180,E1 -19141.91,E2 -19141.91} C_VEL
LIN {X 0,Y 256.475,Z 314.976,A -85,B 0,C 180,E1 -19142.568,E2 -19142.568} C_VEL
LIN {X 0,Y 254.755,Z 326.787,A -85,B 0,C 180,E1 -19143.587,E2 -19143.587} C_VEL
LIN {X 0,Y 252.768,Z 338.183,A -85,B 0,C 180,E1 -19144.912,E2 -19144.912} C_VEL
LIN {X 0,Y 250.609,Z 348.475,A -85,B 0,C 180,E1 -19146.446,E2 -19146.446} C_VEL
LIN {X 0,Y 248.643,Z 356.999,A -85,B 0,C 180,E1 -19148.006,E2 -19148.006} C_VEL
LIN {X 0,Y 246.98,Z 364.218,A -85,B 0,C 180,E1 -19149.6,E2 -19149.6} C_VEL
LIN {X 0,Y 245.621,Z 370.284,A -85,B 0,C 180,E1 -19151.179,E2 -19151.179} C_VEL
LIN {X 0,Y 243.923,Z 376.957,A -85,B 0,C 180,E1 -19153.255,E2 -19153.255} C_VEL
LIN {X 0,Y 242.811,Z 381.459,A -85,B 0,C 180,E1 -19154.9,E2 -19154.9} C_VEL
LIN {X 0,Y 241.462,Z 386.95,A -85,B 0,C 180,E1 -19157.391,E2 -19157.391} C_VEL
LIN {X 0,Y 240.603,Z 391.279,A -85,B 0,C 180,E1 -19159.906,E2 -19159.906} C_VEL
LIN {X 0,Y 240.209,Z 393.648,A -85,B 0,C 180,E1 -19161.588,E2 -19161.588} C_VEL
LIN {X 0,Y 239.928,Z 395.45,A -85,B 0,C 180,E1 -19163.271,E2 -19163.271} C_VEL
LIN {X 0,Y 239.764,Z 397.903,A -85,B 0,C 180,E1 -19166.639,E2 -19166.639} C_VEL
LIN {X 0,Y 239.816,Z 398.496,A -85,B 0,C 180,E1 -19168.321,E2 -19168.321} C_VEL
LIN {X 0,Y 239.884,Z 398.653,A -85,B 0,C 180,E1 -19170,E2 -19170} C_VEL
LIN {X 0,Y 239.816,Z 398.496,A -85,B 0,C 180,E1 -19171.679,E2 -19171.679} C_VEL
LIN {X 0,Y 239.761,Z 397.903,A -85,B 0,C 180,E1 -19173.361,E2 -19173.361} C_VEL
LIN {X 0,Y 239.908,Z 395.449,A -85,B 0,C 180,E1 -19176.729,E2 -19176.729} C_VEL
LIN {X 0,Y 240.378,Z 392.497,A -85,B 0,C 180,E1 -19179.254,E2 -19179.254} C_VEL
LIN {X 0,Y 241.149,Z 388.505,A -85,B 0,C 180,E1 -19181.771,E2 -19181.771} C_VEL
LIN {X 0,Y 242.288,Z 383.373,A -85,B 0,C 180,E1 -19184.274,E2 -19184.274} C_VEL
LIN {X 0,Y 243.667,Z 378.114,A -85,B 0,C 180,E1 -19186.333,E2 -19186.333} C_VEL
LIN {X 0,Y 245.235,Z 371.798,A -85,B 0,C 180,E1 -19188.375,E2 -19188.375} C_VEL
LIN {X 0,Y 246.637,Z 365.846,A -85,B 0,C 180,E1 -19189.995,E2 -19189.995} C_VEL
LIN {X 0,Y 248.201,Z 358.918,A -85,B 0,C 180,E1 -19191.599,E2 -19191.599} C_VEL
LIN {X 0,Y 250.084,Z 350.742,A -85,B 0,C 180,E1 -19193.168,E2 -19193.168} C_VEL
LIN {X 0,Y 251.908,Z 342.234,A -85,B 0,C 180,E1 -19194.519,E2 -19194.519} C_VEL
LIN {X 0,Y 253.611,Z 333.523,A -85,B 0,C 180,E1 -19195.658,E2 -19195.658} C_VEL
LIN {X 0,Y 255.237,Z 323.768,A -85,B 0,C 180,E1 -19196.69,E2 -19196.69} C_VEL
LIN {X 0,Y 256.613,Z 313.688,A -85,B 0,C 180,E1 -19197.527,E2 -19197.527} C_VEL
LIN {X 0,Y 257.768,Z 303.814,A -85,B 0,C 180,E1 -19198.133,E2 -19198.133} C_VEL
LIN {X 0,Y 258.544,Z 294.09,A -85,B 0,C 180,E1 -19198.562,E2 -19198.562} C_VEL
LIN {X 0,Y 260.432,Z 241.559,A -85,B 0,C 180,E1 -19200.017,E2 -19200.017} C_VEL
LIN {X 0,Y 257.935,Z 225.978,A -85,B 0,C 180,E1 -19200.828,E2 -19200.828} C_VEL
LIN {X 0,Y 254.835,Z 210.73,A -85,B 0,C 180,E1 -19201.735,E2 -19201.735} C_VEL
LIN {X 0,Y 247.689,Z 194.529,A -85,B 0,C 180,E1 -19203.303,E2 -19203.303} C_VEL
LIN {X 0,Y 244.646,Z 187.913,A -85,B 0,C 180,E1 -19204.036,E2 -19204.036} C_VEL
LIN {X 0,Y 244.337,Z 186.619,A -85,B 0,C 180,E1 -19204.507,E2 -19204.507} C_VEL
LIN {X 0,Y 242.831,Z 179.305,A -85,B 0,C 180,E1 -19208.607,E2 -19208.607} C_VEL
LIN {X 0,Y 241.994,Z 175.9,A -85,B 0,C 180,E1 -19210.669,E2 -19210.669} C_VEL
LIN {X 0,Y 241.927,Z 175.844,A -85,B 0,C 180,E1 -19214.202,E2 -19214.202} C_VEL
LIN {X 0,Y 241.935,Z 175.847,A -85,B 0,C 180,E1 -19218.076,E2 -19218.076} C_VEL
LIN {X 0,Y 241.995,Z 175.841,A -85,B 0,C 180,E1 -19222.418,E2 -19222.418} C_VEL
LIN {X 0,Y 241.982,Z 175.818,A -85,B 0,C 180,E1 -19226.507,E2 -19226.507} C_VEL
LIN {X 0,Y 242.036,Z 175.827,A -85,B 0,C 180,E1 -19230.587,E2 -19230.587} C_VEL
LIN {X 0,Y 242.068,Z 175.804,A -85,B 0,C 180,E1 -19234.182,E2 -19234.182} C_VEL
LIN {X 0,Y 242.053,Z 175.824,A -85,B 0,C 180,E1 -19238.296,E2 -19238.296} C_VEL
LIN {X 0,Y 242.163,Z 175.795,A -85,B 0,C 180,E1 -19243.277,E2 -19243.277} C_VEL
LIN {X 0,Y 242.18,Z 175.791,A -85,B 0,C 180,E1 -19248.279,E2 -19248.279} C_VEL
LIN {X 0,Y 242.399,Z 175.752,A -85,B 0,C 180,E1 -19251.664,E2 -19251.664} C_VEL
LIN {X 0,Y 242.256,Z 175.809,A -85,B 0,C 180,E1 -19255.006,E2 -19255.006} C_VEL
LIN {X 0,Y 242.634,Z 175.73,A -85,B 0,C 180,E1 -19258.339,E2 -19258.339} C_VEL
LIN {X 0,Y 242.635,Z 175.725,A -85,B 0,C 180,E1 -19261.659,E2 -19261.659} C_VEL
LIN {X 0,Y 242.428,Z 175.778,A -85,B 0,C 180,E1 -19266.706,E2 -19266.706} C_VEL
LIN {X 0,Y 242.312,Z 175.757,A -85,B 0,C 180,E1 -19270.021,E2 -19270.021} C_VEL
LIN {X 0,Y 242.164,Z 175.819,A -85,B 0,C 180,E1 -19275.14,E2 -19275.14} C_VEL
LIN {X 0,Y 242.07,Z 175.792,A -85,B 0,C 180,E1 -19278.623,E2 -19278.623} C_VEL
LIN {X 0,Y 242.01,Z 175.833,A -85,B 0,C 180,E1 -19282.179,E2 -19282.179} C_VEL
LIN {X 0,Y 242.063,Z 175.81,A -85,B 0,C 180,E1 -19285.837,E2 -19285.837} C_VEL
LIN {X 0,Y 242.027,Z 175.827,A -85,B 0,C 180,E1 -19289.579,E2 -19289.579} C_VEL
LIN {X 0,Y 241.988,Z 175.819,A -85,B 0,C 180,E1 -19293.49,E2 -19293.49} C_VEL
LIN {X 0,Y 241.999,Z 175.844,A -85,B 0,C 180,E1 -19297.579,E2 -19297.579} C_VEL
LIN {X 0,Y 241.94,Z 175.835,A -85,B 0,C 180,E1 -19301.92,E2 -19301.92} C_VEL
LIN {X 0,Y 241.932,Z 175.793,A -85,B 0,C 180,E1 -19306.57,E2 -19306.57} C_VEL
LIN {X 0,Y 241.968,Z 175.806,A -85,B 0,C 180,E1 -19310.284,E2 -19310.284} C_VEL
LIN {X 0,Y 242.033,Z 175.799,A -85,B 0,C 180,E1 -19314.497,E2 -19314.497} C_VEL
LIN {X 0,Y 242.076,Z 176.073,A -85,B 0,C 180,E1 -19315.364,E2 -19315.364} C_VEL
LIN {X 0,Y 242.428,Z 177.42,A -85,B 0,C 180,E1 -19315.65,E2 -19315.65} C_VEL
LIN {X 0,Y 251.85,Z 193.897,A -85,B 0,C 180,E1 -19317.671,E2 -19317.671} C_VEL
LIN {X 0,Y 261.766,Z 212.756,A -85,B 0,C 180,E1 -19319.635,E2 -19319.635} C_VEL
LIN {X 0,Y 269.822,Z 224.726,A -85,B 0,C 180,E1 -19320.998,E2 -19320.998} C_VEL
LIN {X 0,Y 279.916,Z 236.888,A -85,B 0,C 180,E1 -19322.492,E2 -19322.492} C_VEL
LIN {X 0,Y 294.711,Z 251.776,A -85,B 0,C 180,E1 -19324.387,E2 -19324.387} C_VEL
LIN {X 0,Y 306.273,Z 261.77,A -85,B 0,C 180,E1 -19325.791,E2 -19325.791} C_VEL
LIN {X 0,Y 315.078,Z 269.134,A -85,B 0,C 180,E1 -19327.073,E2 -19327.073} C_VEL
LIN {X 0,Y 322.662,Z 275.113,A -85,B 0,C 180,E1 -19328.331,E2 -19328.331} C_VEL
LIN {X 0,Y 329.947,Z 280.607,A -85,B 0,C 180,E1 -19329.705,E2 -19329.705} C_VEL
LIN {X 0,Y 338.471,Z 287.031,A -85,B 0,C 180,E1 -19331.517,E2 -19331.517} C_VEL
LIN {X 0,Y 346.337,Z 292.474,A -85,B 0,C 180,E1 -19333.405,E2 -19333.405} C_VEL
LIN {X 0,Y 352.216,Z 296.745,A -85,B 0,C 180,E1 -19335.01,E2 -19335.01} C_VEL
LIN {X 0,Y 357.969,Z 300.283,A -85,B 0,C 180,E1 -19336.773,E2 -19336.773} C_VEL
LIN {X 0,Y 361.254,Z 302.277,A -85,B 0,C 180,E1 -19337.912,E2 -19337.912} C_VEL
LIN {X 0,Y 365.801,Z 305.72,A -85,B 0,C 180,E1 -19339.774,E2 -19339.774} C_VEL
LIN {X 0,Y 369.469,Z 308.038,A -85,B 0,C 180,E1 -19341.542,E2 -19341.542} C_VEL
LIN {X 0,Y 372.788,Z 309.755,A -85,B 0,C 180,E1 -19343.505,E2 -19343.505} C_VEL
LIN {X 0,Y 374.917,Z 310.696,A -85,B 0,C 180,E1 -19345.169,E2 -19345.169} C_VEL
LIN {X 0,Y 376.633,Z 311.22,A -85,B 0,C 180,E1 -19347.059,E2 -19347.059} C_VEL
LIN {X 0,Y 377.443,Z 311.735,A -85,B 0,C 180,E1 -19348.933,E2 -19348.933} C_VEL
LIN {X 0,Y 377.606,Z 311.662,A -85,B 0,C 180,E1 -19350,E2 -19350} C_VEL
LIN {X 0,Y 377.309,Z 311.605,A -85,B 0,C 180,E1 -19351.601,E2 -19351.601} C_VEL
LIN {X 0,Y 376.471,Z 311.092,A -85,B 0,C 180,E1 -19353.21,E2 -19353.21} C_VEL
LIN {X 0,Y 374.606,Z 310.544,A -85,B 0,C 180,E1 -19355.11,E2 -19355.11} C_VEL
LIN {X 0,Y 371.87,Z 309.318,A -85,B 0,C 180,E1 -19357.085,E2 -19357.085} C_VEL
LIN {X 0,Y 368.482,Z 307.458,A -85,B 0,C 180,E1 -19358.951,E2 -19358.951} C_VEL
LIN {X 0,Y 364.539,Z 304.862,A -85,B 0,C 180,E1 -19360.759,E2 -19360.759} C_VEL
LIN {X 0,Y 359.989,Z 301.382,A -85,B 0,C 180,E1 -19362.544,E2 -19362.544} C_VEL
LIN {X 0,Y 354.625,Z 298.331,A -85,B 0,C 180,E1 -19364.272,E2 -19364.272} C_VEL
LIN {X 0,Y 348.535,Z 294.17,A -85,B 0,C 180,E1 -19366.012,E2 -19366.012} C_VEL
LIN {X 0,Y 342.479,Z 289.746,A -85,B 0,C 180,E1 -19367.556,E2 -19367.556} C_VEL
LIN {X 0,Y 335.425,Z 284.797,A -85,B 0,C 180,E1 -19369.152,E2 -19369.152} C_VEL
LIN {X 0,Y 328.365,Z 279.467,A -85,B 0,C 180,E1 -19370.607,E2 -19370.607} C_VEL
LIN {X 0,Y 321.234,Z 273.929,A -85,B 0,C 180,E1 -19371.923,E2 -19371.923} C_VEL
LIN {X 0,Y 311.861,Z 266.525,A -85,B 0,C 180,E1 -19373.421,E2 -19373.421} C_VEL
LIN {X 0,Y 302.673,Z 258.796,A -85,B 0,C 180,E1 -19374.662,E2 -19374.662} C_VEL
LIN {X 0,Y 290.463,Z 247.675,A -85,B 0,C 180,E1 -19376.13,E2 -19376.13} C_VEL
LIN {X 0,Y 277.867,Z 234.573,A -85,B 0,C 180,E1 -19377.797,E2 -19377.797} C_VEL
LIN {X 0,Y 269.468,Z 224.243,A -85,B 0,C 180,E1 -19379.059,E2 -19379.059} C_VEL
LIN {X 0,Y 261.201,Z 211.814,A -85,B 0,C 180,E1 -19380.468,E2 -19380.468} C_VEL
LIN {X 0,Y 249.278,Z 189.349,A -85,B 0,C 180,E1 -19382.859,E2 -19382.859} C_VEL
LIN {X 0,Y 243.309,Z 179.091,A -85,B 0,C 180,E1 -19384.137,E2 -19384.137} C_VEL
LIN {X 0,Y 242.164,Z 176.522,A -85,B 0,C 180,E1 -19384.492,E2 -19384.492} C_VEL
LIN {X 0,Y 242.025,Z 175.847,A -85,B 0,C 180,E1 -19384.936,E2 -19384.936} C_VEL
LIN {X 0,Y 242.003,Z 175.839,A -85,B 0,C 180,E1 -19388.364,E2 -19388.364} C_VEL
LIN {X 0,Y 241.94,Z 175.784,A -85,B 0,C 180,E1 -19391.921,E2 -19391.921} C_VEL
LIN {X 0,Y 241.933,Z 175.85,A -85,B 0,C 180,E1 -19396.571,E2 -19396.571} C_VEL
LIN {X 0,Y 241.968,Z 175.828,A -85,B 0,C 180,E1 -19400.285,E2 -19400.285} C_VEL
LIN {X 0,Y 242.033,Z 175.814,A -85,B 0,C 180,E1 -19404.498,E2 -19404.498} C_VEL
LIN {X 0,Y 241.973,Z 175.845,A -85,B 0,C 180,E1 -19408.481,E2 -19408.481} C_VEL
LIN {X 0,Y 242.005,Z 175.808,A -85,B 0,C 180,E1 -19412.313,E2 -19412.313} C_VEL
LIN {X 0,Y 242.054,Z 175.832,A -85,B 0,C 180,E1 -19416.017,E2 -19416.017} C_VEL
LIN {X 0,Y 242.034,Z 175.804,A -85,B 0,C 180,E1 -19419.609,E2 -19419.609} C_VEL
LIN {X 0,Y 242.161,Z 175.803,A -85,B 0,C 180,E1 -19423.279,E2 -19423.279} C_VEL
LIN {X 0,Y 242.184,Z 175.789,A -85,B 0,C 180,E1 -19428.281,E2 -19428.281} C_VEL
LIN {X 0,Y 242.426,Z 175.754,A -85,B 0,C 180,E1 -19431.666,E2 -19431.666} C_VEL
LIN {X 0,Y 242.259,Z 175.808,A -85,B 0,C 180,E1 -19435.008,E2 -19435.008} C_VEL
LIN {X 0,Y 242.635,Z 175.725,A -85,B 0,C 180,E1 -19438.341,E2 -19438.341} C_VEL
LIN {X 0,Y 242.634,Z 175.73,A -85,B 0,C 180,E1 -19441.661,E2 -19441.661} C_VEL
LIN {X 0,Y 242.422,Z 175.775,A -85,B 0,C 180,E1 -19446.66,E2 -19446.66} C_VEL
LIN {X 0,Y 242.266,Z 175.762,A -85,B 0,C 180,E1 -19450.025,E2 -19450.025} C_VEL
LIN {X 0,Y 242.166,Z 175.814,A -85,B 0,C 180,E1 -19455.142,E2 -19455.142} C_VEL
LIN {X 0,Y 242.072,Z 175.789,A -85,B 0,C 180,E1 -19458.625,E2 -19458.625} C_VEL
LIN {X 0,Y 242.013,Z 175.834,A -85,B 0,C 180,E1 -19462.181,E2 -19462.181} C_VEL
LIN {X 0,Y 242.067,Z 175.803,A -85,B 0,C 180,E1 -19465.839,E2 -19465.839} C_VEL
LIN {X 0,Y 242.029,Z 175.83,A -85,B 0,C 180,E1 -19469.581,E2 -19469.581} C_VEL
LIN {X 0,Y 241.982,Z 175.818,A -85,B 0,C 180,E1 -19473.493,E2 -19473.493} C_VEL
LIN {X 0,Y 241.995,Z 175.841,A -85,B 0,C 180,E1 -19477.582,E2 -19477.582} C_VEL
LIN {X 0,Y 241.934,Z 175.846,A -85,B 0,C 180,E1 -19481.924,E2 -19481.924} C_VEL
LIN {X 0,Y 241.934,Z 175.852,A -85,B 0,C 180,E1 -19486.573,E2 -19486.573} C_VEL
LIN {X 0,Y 242.024,Z 175.978,A -85,B 0,C 180,E1 -19489.423,E2 -19489.423} C_VEL
LIN {X 0,Y 243.608,Z 182.794,A -85,B 0,C 180,E1 -19493.382,E2 -19493.382} C_VEL
LIN {X 0,Y 244.164,Z 185.696,A -85,B 0,C 180,E1 -19494.995,E2 -19494.995} C_VEL
LIN {X 0,Y 244.755,Z 187.83,A -85,B 0,C 180,E1 -19495.7,E2 -19495.7} C_VEL
LIN {X 0,Y 245.707,Z 190.805,A -85,B 0,C 180,E1 -19496.205,E2 -19496.205} C_VEL
LIN {X 0,Y 247.238,Z 196.147,A -85,B 0,C 180,E1 -19496.684,E2 -19496.684} C_VEL
LIN {X 0,Y 248.474,Z 206.422,A -85,B 0,C 180,E1 -19497.203,E2 -19497.203} C_VEL
LIN {X 0,Y 249.416,Z 214.768,A -85,B 0,C 180,E1 -19497.633,E2 -19497.633} C_VEL
LIN {X 0,Y 253.13,Z 234.628,A -85,B 0,C 180,E1 -19498.806,E2 -19498.806} C_VEL
LIN {X 0,Y 254.258,Z 242.726,A -85,B 0,C 180,E1 -19499.219,E2 -19499.219} C_VEL
LIN {X 0,Y 252.388,Z 293.303,A -85,B 0,C 180,E1 -19500.646,E2 -19500.646} C_VEL
LIN {X 0,Y 251.509,Z 303.806,A -85,B 0,C 180,E1 -19501.114,E2 -19501.114} C_VEL
LIN {X 0,Y 250.36,Z 313.497,A -85,B 0,C 180,E1 -19501.725,E2 -19501.725} C_VEL
LIN {X 0,Y 248.901,Z 323.576,A -85,B 0,C 180,E1 -19502.574,E2 -19502.574} C_VEL
LIN {X 0,Y 247.255,Z 333.332,A -85,B 0,C 180,E1 -19503.633,E2 -19503.633} C_VEL
LIN {X 0,Y 245.183,Z 343.394,A -85,B 0,C 180,E1 -19504.989,E2 -19504.989} C_VEL
LIN {X 0,Y 242.561,Z 354.889,A -85,B 0,C 180,E1 -19506.974,E2 -19506.974} C_VEL
LIN {X 0,Y 240.299,Z 364.025,A -85,B 0,C 180,E1 -19509.006,E2 -19509.006} C_VEL
LIN {X 0,Y 238.791,Z 370.402,A -85,B 0,C 180,E1 -19510.72,E2 -19510.72} C_VEL
LIN {X 0,Y 237.082,Z 376.764,A -85,B 0,C 180,E1 -19512.756,E2 -19512.756} C_VEL
LIN {X 0,Y 235.932,Z 381.266,A -85,B 0,C 180,E1 -19514.449,E2 -19514.449} C_VEL
LIN {X 0,Y 234.507,Z 386.758,A -85,B 0,C 180,E1 -19517.011,E2 -19517.011} C_VEL
LIN {X 0,Y 233.577,Z 391.086,A -85,B 0,C 180,E1 -19519.599,E2 -19519.599} C_VEL
LIN {X 0,Y 233.177,Z 393.457,A -85,B 0,C 180,E1 -19521.333,E2 -19521.333} C_VEL
LIN {X 0,Y 232.874,Z 395.258,A -85,B 0,C 180,E1 -19523.067,E2 -19523.067} C_VEL
LIN {X 0,Y 232.674,Z 397.711,A -85,B 0,C 180,E1 -19526.537,E2 -19526.537} C_VEL
LIN {X 0,Y 232.729,Z 398.304,A -85,B 0,C 180,E1 -19528.27,E2 -19528.27} C_VEL
LIN {X 0,Y 232.795,Z 398.461,A -85,B 0,C 180,E1 -19530,E2 -19530} C_VEL
LIN {X 0,Y 232.729,Z 398.304,A -85,B 0,C 180,E1 -19531.73,E2 -19531.73} C_VEL
LIN {X 0,Y 232.689,Z 397.033,A -85,B 0,C 180,E1 -19534.637,E2 -19534.637} C_VEL
LIN {X 0,Y 232.83,Z 395.257,A -85,B 0,C 180,E1 -19536.935,E2 -19536.935} C_VEL
LIN {X 0,Y 233.362,Z 392.305,A -85,B 0,C 180,E1 -19539.534,E2 -19539.534} C_VEL
LIN {X 0,Y 234.164,Z 388.313,A -85,B 0,C 180,E1 -19542.128,E2 -19542.128} C_VEL
LIN {X 0,Y 235.391,Z 383.181,A -85,B 0,C 180,E1 -19544.701,E2 -19544.701} C_VEL
LIN {X 0,Y 236.834,Z 377.921,A -85,B 0,C 180,E1 -19546.818,E2 -19546.818} C_VEL
LIN {X 0,Y 238.477,Z 371.605,A -85,B 0,C 180,E1 -19548.915,E2 -19548.915} C_VEL
LIN {X 0,Y 239.94,Z 365.653,A -85,B 0,C 180,E1 -19550.578,E2 -19550.578} C_VEL
LIN {X 0,Y 241.604,Z 358.726,A -85,B 0,C 180,E1 -19552.219,E2 -19552.219} C_VEL
LIN {X 0,Y 243.57,Z 350.55,A -85,B 0,C 180,E1 -19553.826,E2 -19553.826} C_VEL
LIN {X 0,Y 245.448,Z 342.042,A -85,B 0,C 180,E1 -19555.209,E2 -19555.209} C_VEL
LIN {X 0,Y 247.216,Z 333.331,A -85,B 0,C 180,E1 -19556.372,E2 -19556.372} C_VEL
LIN {X 0,Y 248.907,Z 323.576,A -85,B 0,C 180,E1 -19557.425,E2 -19557.425} C_VEL
LIN {X 0,Y 250.352,Z 313.497,A -85,B 0,C 180,E1 -19558.276,E2 -19558.276} C_VEL
LIN {X 0,Y 251.511,Z 303.839,A -85,B 0,C 180,E1 -19558.884,E2 -19558.884} C_VEL
LIN {X 0,Y 252.295,Z 294.558,A -85,B 0,C 180,E1 -19559.309,E2 -19559.309} C_VEL
LIN {X 0,Y 253.491,Z 263.676,A -85,B 0,C 180,E1 -19560.209,E2 -19560.209} C_VEL
LIN {X 0,Y 254.211,Z 241.515,A -85,B 0,C 180,E1 -19560.826,E2 -19560.826} C_VEL
LIN {X 0,Y 250.672,Z 221.043,A -85,B 0,C 180,E1 -19561.979,E2 -19561.979} C_VEL
LIN {X 0,Y 248.998,Z 213.275,A -85,B 0,C 180,E1 -19562.478,E2 -19562.478} C_VEL
LIN {X 0,Y 242.23,Z 197.858,A -85,B 0,C 180,E1 -19564.033,E2 -19564.033} C_VEL
LIN {X 0,Y 237.347,Z 187.572,A -85,B 0,C 180,E1 -19565.251,E2 -19565.251} C_VEL
LIN {X 0,Y 236.76,Z 184.625,A -85,B 0,C 180,E1 -19566.728,E2 -19566.728} C_VEL
LIN {X 0,Y 235.382,Z 178.702,A -85,B 0,C 180,E1 -19570.272,E2 -19570.272} C_VEL
LIN {X 0,Y 234.919,Z 176.733,A -85,B 0,C 180,E1 -19571.589,E2 -19571.589} C_VEL
LIN {X 0,Y 234.889,Z 176.716,A -85,B 0,C 180,E1 -19575.897,E2 -19575.897} C_VEL
LIN {X 0,Y 234.882,Z 176.715,A -85,B 0,C 180,E1 -19578.831,E2 -19578.831} C_VEL
LIN {X 0,Y 234.92,Z 176.71,A -85,B 0,C 180,E1 -19581.078,E2 -19581.078} C_VEL
LIN {X 0,Y 234.934,Z 176.694,A -85,B 0,C 180,E1 -19585.362,E2 -19585.362} C_VEL
LIN {X 0,Y 234.932,Z 176.721,A -85,B 0,C 180,E1 -19589.431,E2 -19589.431} C_VEL
LIN {X 0,Y 234.994,Z 176.681,A -85,B 0,C 180,E1 -19593.793,E2 -19593.793} C_VEL
LIN {X 0,Y 235.011,Z 176.692,A -85,B 0,C 180,E1 -19598.969,E2 -19598.969} C_VEL
LIN {X 0,Y 235.096,Z 176.671,A -85,B 0,C 180,E1 -19603.059,E2 -19603.059} C_VEL
LIN {X 0,Y 235.114,Z 176.675,A -85,B 0,C 180,E1 -19607.921,E2 -19607.921} C_VEL
LIN {X 0,Y 235.33,Z 176.629,A -85,B 0,C 180,E1 -19611.411,E2 -19611.411} C_VEL
LIN {X 0,Y 235.372,Z 176.649,A -85,B 0,C 180,E1 -19613.14,E2 -19613.14} C_VEL
LIN {X 0,Y 235.593,Z 176.607,A -85,B 0,C 180,E1 -19618.29,E2 -19618.29} C_VEL
LIN {X 0,Y 235.594,Z 176.602,A -85,B 0,C 180,E1 -19621.709,E2 -19621.709} C_VEL
LIN {X 0,Y 235.402,Z 176.651,A -85,B 0,C 180,E1 -19626.858,E2 -19626.858} C_VEL
LIN {X 0,Y 235.236,Z 176.639,A -85,B 0,C 180,E1 -19630.326,E2 -19630.326} C_VEL
LIN {X 0,Y 235.111,Z 176.695,A -85,B 0,C 180,E1 -19635.606,E2 -19635.606} C_VEL
LIN {X 0,Y 235.005,Z 176.67,A -85,B 0,C 180,E1 -19639.205,E2 -19639.205} C_VEL
LIN {X 0,Y 234.958,Z 176.717,A -85,B 0,C 180,E1 -19642.882,E2 -19642.882} C_VEL
LIN {X 0,Y 234.967,Z 176.685,A -85,B 0,C 180,E1 -19646.657,E2 -19646.657} C_VEL
LIN {X 0,Y 234.929,Z 176.722,A -85,B 0,C 180,E1 -19650.567,E2 -19650.567} C_VEL
LIN {X 0,Y 234.957,Z 176.69,A -85,B 0,C 180,E1 -19654.632,E2 -19654.632} C_VEL
LIN {X 0,Y 234.938,Z 176.712,A -85,B 0,C 180,E1 -19658.944,E2 -19658.944} C_VEL
LIN {X 0,Y 234.886,Z 176.727,A -85,B 0,C 180,E1 -19663.485,E2 -19663.485} C_VEL
LIN {X 0,Y 234.885,Z 176.67,A -85,B 0,C 180,E1 -19666.514,E2 -19666.514} C_VEL
LIN {X 0,Y 234.951,Z 176.698,A -85,B 0,C 180,E1 -19671.086,E2 -19671.086} C_VEL
LIN {X 0,Y 235.006,Z 176.925,A -85,B 0,C 180,E1 -19674.156,E2 -19674.156} C_VEL
LIN {X 0,Y 235.26,Z 177.882,A -85,B 0,C 180,E1 -19674.444,E2 -19674.444} C_VEL
LIN {X 0,Y 236.738,Z 180.558,A -85,B 0,C 180,E1 -19674.823,E2 -19674.823} C_VEL
LIN {X 0,Y 245.37,Z 195.609,A -85,B 0,C 180,E1 -19676.76,E2 -19676.76} C_VEL
LIN {X 0,Y 257.214,Z 217.96,A -85,B 0,C 180,E1 -19679.201,E2 -19679.201} C_VEL
LIN {X 0,Y 265.912,Z 230.814,A -85,B 0,C 180,E1 -19680.711,E2 -19680.711} C_VEL
LIN {X 0,Y 277.032,Z 243.819,A -85,B 0,C 180,E1 -19682.377,E2 -19682.377} C_VEL
LIN {X 0,Y 290.947,Z 257.725,A -85,B 0,C 180,E1 -19684.188,E2 -19684.188} C_VEL
LIN {X 0,Y 302.696,Z 267.809,A -85,B 0,C 180,E1 -19685.584,E2 -19685.584} C_VEL
LIN {X 0,Y 312.33,Z 275.676,A -85,B 0,C 180,E1 -19686.889,E2 -19686.889} C_VEL
LIN {X 0,Y 320.422,Z 281.999,A -85,B 0,C 180,E1 -19688.21,E2 -19688.21} C_VEL
LIN {X 0,Y 328.313,Z 287.748,A -85,B 0,C 180,E1 -19689.685,E2 -19689.685} C_VEL
LIN {X 0,Y 336.055,Z 293.62,A -85,B 0,C 180,E1 -19691.33,E2 -19691.33} C_VEL
LIN {X 0,Y 343.932,Z 299.027,A -85,B 0,C 180,E1 -19693.204,E2 -19693.204} C_VEL
LIN {X 0,Y 350.177,Z 303.568,A -85,B 0,C 180,E1 -19694.92,E2 -19694.92} C_VEL
LIN {X 0,Y 356.042,Z 307.136,A -85,B 0,C 180,E1 -19696.718,E2 -19696.718} C_VEL
LIN {X 0,Y 359.401,Z 309.2,A -85,B 0,C 180,E1 -19697.884,E2 -19697.884} C_VEL
LIN {X 0,Y 363.782,Z 312.48,A -85,B 0,C 180,E1 -19699.69,E2 -19699.69} C_VEL
LIN {X 0,Y 366.921,Z 314.483,A -85,B 0,C 180,E1 -19701.186,E2 -19701.186} C_VEL
LIN {X 0,Y 369.056,Z 315.681,A -85,B 0,C 180,E1 -19702.34,E2 -19702.34} C_VEL
LIN {X 0,Y 370.862,Z 316.569,A -85,B 0,C 180,E1 -19703.471,E2 -19703.471} C_VEL
LIN {X 0,Y 372.383,Z 317.224,A -85,B 0,C 180,E1 -19704.585,E2 -19704.585} C_VEL
LIN {X 0,Y 373.636,Z 317.667,A -85,B 0,C 180,E1 -19705.685,E2 -19705.685} C_VEL
LIN {X 0,Y 374.612,Z 317.952,A -85,B 0,C 180,E1 -19706.774,E2 -19706.774} C_VEL
LIN {X 0,Y 375.245,Z 318.321,A -85,B 0,C 180,E1 -19707.853,E2 -19707.853} C_VEL
LIN {X 0,Y 375.607,Z 318.593,A -85,B 0,C 180,E1 -19708.928,E2 -19708.928} C_VEL
LIN {X 0,Y 375.785,Z 318.503,A -85,B 0,C 180,E1 -19710,E2 -19710} C_VEL
LIN {X 0,Y 375.629,Z 318.529,A -85,B 0,C 180,E1 -19711.072,E2 -19711.072} C_VEL
LIN {X 0,Y 375.258,Z 318.298,A -85,B 0,C 180,E1 -19712.147,E2 -19712.147} C_VEL
LIN {X 0,Y 374.622,Z 317.947,A -85,B 0,C 180,E1 -19713.226,E2 -19713.226} C_VEL
LIN {X 0,Y 373.577,Z 317.648,A -85,B 0,C 180,E1 -19714.394,E2 -19714.394} C_VEL
LIN {X 0,Y 372.402,Z 317.239,A -85,B 0,C 180,E1 -19715.414,E2 -19715.414} C_VEL
LIN {X 0,Y 370.877,Z 316.583,A -85,B 0,C 180,E1 -19716.528,E2 -19716.528} C_VEL
LIN {X 0,Y 368.834,Z 315.571,A -85,B 0,C 180,E1 -19717.767,E2 -19717.767} C_VEL
LIN {X 0,Y 365.354,Z 313.544,A -85,B 0,C 180,E1 -19719.585,E2 -19719.585} C_VEL
LIN {X 0,Y 361.254,Z 310.665,A -85,B 0,C 180,E1 -19721.37,E2 -19721.37} C_VEL
LIN {X 0,Y 357.701,Z 308.023,A -85,B 0,C 180,E1 -19722.733,E2 -19722.733} C_VEL
LIN {X 0,Y 351.866,Z 304.653,A -85,B 0,C 180,E1 -19724.58,E2 -19724.58} C_VEL
LIN {X 0,Y 345.803,Z 300.495,A -85,B 0,C 180,E1 -19726.29,E2 -19726.29} C_VEL
LIN {X 0,Y 339.864,Z 296.239,A -85,B 0,C 180,E1 -19727.788,E2 -19727.788} C_VEL
LIN {X 0,Y 332.543,Z 291.079,A -85,B 0,C 180,E1 -19729.436,E2 -19729.436} C_VEL
LIN {X 0,Y 325.158,Z 285.521,A -85,B 0,C 180,E1 -19730.922,E2 -19730.922} C_VEL
LIN {X 0,Y 317.749,Z 279.824,A -85,B 0,C 180,E1 -19732.254,E2 -19732.254} C_VEL
LIN {X 0,Y 309.982,Z 273.876,A -85,B 0,C 180,E1 -19733.436,E2 -19733.436} C_VEL
LIN {X 0,Y 301.951,Z 267.178,A -85,B 0,C 180,E1 -19734.508,E2 -19734.508} C_VEL
LIN {X 0,Y 290.543,Z 257.362,A -85,B 0,C 180,E1 -19735.861,E2 -19735.861} C_VEL
LIN {X 0,Y 275.739,Z 242.485,A -85,B 0,C 180,E1 -19737.803,E2 -19737.803} C_VEL
LIN {X 0,Y 265.573,Z 230.305,A -85,B 0,C 180,E1 -19739.346,E2 -19739.346} C_VEL
LIN {X 0,Y 257.557,Z 218.504,A -85,B 0,C 180,E1 -19740.736,E2 -19740.736} C_VEL
LIN {X 0,Y 250.53,Z 205.561,A -85,B 0,C 180,E1 -19742.133,E2 -19742.133} C_VEL
LIN {X 0,Y 244.32,Z 193.683,A -85,B 0,C 180,E1 -19743.469,E2 -19743.469} C_VEL
LIN {X 0,Y 236.565,Z 180.35,A -85,B 0,C 180,E1 -19745.214,E2 -19745.214} C_VEL
LIN {X 0,Y 235.13,Z 177.427,A -85,B 0,C 180,E1 -19745.648,E2 -19745.648} C_VEL
LIN {X 0,Y 234.952,Z 176.731,A -85,B 0,C 180,E1 -19746.136,E2 -19746.136} C_VEL
LIN {X 0,Y 234.938,Z 176.698,A -85,B 0,C 180,E1 -19748.945,E2 -19748.945} C_VEL
LIN {X 0,Y 234.885,Z 176.67,A -85,B 0,C 180,E1 -19753.486,E2 -19753.486} C_VEL
LIN {X 0,Y 234.886,Z 176.727,A -85,B 0,C 180,E1 -19756.515,E2 -19756.515} C_VEL
LIN {X 0,Y 234.951,Z 176.71,A -85,B 0,C 180,E1 -19761.087,E2 -19761.087} C_VEL
LIN {X 0,Y 234.957,Z 176.69,A -85,B 0,C 180,E1 -19765.368,E2 -19765.368} C_VEL
LIN {X 0,Y 234.966,Z 176.709,A -85,B 0,C 180,E1 -19770.158,E2 -19770.158} C_VEL
LIN {X 0,Y 234.991,Z 176.685,A -85,B 0,C 180,E1 -19773.794,E2 -19773.794} C_VEL
LIN {X 0,Y 235.008,Z 176.687,A -85,B 0,C 180,E1 -19778.971,E2 -19778.971} C_VEL
LIN {X 0,Y 235.094,Z 176.678,A -85,B 0,C 180,E1 -19783.06,E2 -19783.06} C_VEL
LIN {X 0,Y 235.144,Z 176.671,A -85,B 0,C 180,E1 -19787.925,E2 -19787.925} C_VEL
LIN {X 0,Y 235.375,Z 176.628,A -85,B 0,C 180,E1 -19791.415,E2 -19791.415} C_VEL
LIN {X 0,Y 235.402,Z 176.651,A -85,B 0,C 180,E1 -19793.142,E2 -19793.142} C_VEL
LIN {X 0,Y 235.594,Z 176.602,A -85,B 0,C 180,E1 -19798.291,E2 -19798.291} C_VEL
LIN {X 0,Y 235.593,Z 176.607,A -85,B 0,C 180,E1 -19801.71,E2 -19801.71} C_VEL
LIN {X 0,Y 235.372,Z 176.649,A -85,B 0,C 180,E1 -19806.86,E2 -19806.86} C_VEL
LIN {X 0,Y 235.213,Z 176.641,A -85,B 0,C 180,E1 -19810.328,E2 -19810.328} C_VEL
LIN {X 0,Y 235.113,Z 176.688,A -85,B 0,C 180,E1 -19815.607,E2 -19815.607} C_VEL
LIN {X 0,Y 235.008,Z 176.669,A -85,B 0,C 180,E1 -19819.207,E2 -19819.207} C_VEL
LIN {X 0,Y 234.961,Z 176.716,A -85,B 0,C 180,E1 -19822.884,E2 -19822.884} C_VEL
LIN {X 0,Y 234.969,Z 176.682,A -85,B 0,C 180,E1 -19826.658,E2 -19826.658} C_VEL
LIN {X 0,Y 234.932,Z 176.721,A -85,B 0,C 180,E1 -19830.569,E2 -19830.569} C_VEL
LIN {X 0,Y 234.934,Z 176.694,A -85,B 0,C 180,E1 -19834.638,E2 -19834.638} C_VEL
LIN {X 0,Y 234.943,Z 176.707,A -85,B 0,C 180,E1 -19838.945,E2 -19838.945} C_VEL
LIN {X 0,Y 234.881,Z 176.721,A -85,B 0,C 180,E1 -19843.488,E2 -19843.488} C_VEL
LIN {X 0,Y 234.897,Z 176.701,A -85,B 0,C 180,E1 -19848.054,E2 -19848.054} C_VEL
LIN {X 0,Y 234.941,Z 176.869,A -85,B 0,C 180,E1 -19848.566,E2 -19848.566} C_VEL
LIN {X 0,Y 236.44,Z 183.195,A -85,B 0,C 180,E1 -19852.428,E2 -19852.428} C_VEL
LIN {X 0,Y 237.307,Z 187.343,A -85,B 0,C 180,E1 -19854.701,E2 -19854.701} C_VEL
LIN {X 0,Y 239.05,Z 191.239,A -85,B 0,C 180,E1 -19855.219,E2 -19855.219} C_VEL
LIN {X 0,Y 246.493,Z 207.24,A -85,B 0,C 180,E1 -19856.949,E2 -19856.949} C_VEL
LIN {X 0,Y 249.416,Z 214.768,A -85,B 0,C 180,E1 -19857.633,E2 -19857.633} C_VEL
LIN {X 0,Y 250.045,Z 220.517,A -85,B 0,C 180,E1 -19857.914,E2 -19857.914} C_VEL
LIN {X 0,Y 249.631,Z 230.331,A -85,B 0,C 180,E1 -19858.18,E2 -19858.18} C_VEL
LIN {X 0,Y 248.06,Z 246.23,A -85,B 0,C 180,E1 -19858.486,E2 -19858.486} C_VEL
LIN {X 0,Y 246.197,Z 293.799,A -85,B 0,C 180,E1 -19859.865,E2 -19859.865} C_VEL
LIN {X 0,Y 245.24,Z 304.622,A -85,B 0,C 180,E1 -19860.371,E2 -19860.371} C_VEL
LIN {X 0,Y 243.808,Z 315.881,A -85,B 0,C 180,E1 -19861.13,E2 -19861.13} C_VEL
LIN {X 0,Y 241.802,Z 328.243,A -85,B 0,C 180,E1 -19862.287,E2 -19862.287} C_VEL
LIN {X 0,Y 239.655,Z 339.149,A -85,B 0,C 180,E1 -19863.67,E2 -19863.67} C_VEL
LIN {X 0,Y 237.614,Z 348.09,A -85,B 0,C 180,E1 -19865.072,E2 -19865.072} C_VEL
LIN {X 0,Y 235.508,Z 356.615,A -85,B 0,C 180,E1 -19866.709,E2 -19866.709} C_VEL
LIN {X 0,Y 233.651,Z 363.832,A -85,B 0,C 180,E1 -19868.379,E2 -19868.379} C_VEL
LIN {X 0,Y 232.238,Z 369.586,A -85,B 0,C 180,E1 -19869.945,E2 -19869.945} C_VEL
LIN {X 0,Y 230.264,Z 376.571,A -85,B 0,C 180,E1 -19872.229,E2 -19872.229} C_VEL
LIN {X 0,Y 229.077,Z 381.074,A -85,B 0,C 180,E1 -19873.972,E2 -19873.972} C_VEL
LIN {X 0,Y 227.545,Z 386.565,A -85,B 0,C 180,E1 -19876.606,E2 -19876.606} C_VEL
LIN {X 0,Y 226.573,Z 390.894,A -85,B 0,C 180,E1 -19879.274,E2 -19879.274} C_VEL
LIN {X 0,Y 226.135,Z 393.264,A -85,B 0,C 180,E1 -19881.06,E2 -19881.06} C_VEL
LIN {X 0,Y 225.811,Z 395.066,A -85,B 0,C 180,E1 -19882.849,E2 -19882.849} C_VEL
LIN {X 0,Y 225.588,Z 397.52,A -85,B 0,C 180,E1 -19886.428,E2 -19886.428} C_VEL
LIN {X 0,Y 225.625,Z 398.113,A -85,B 0,C 180,E1 -19888.215,E2 -19888.215} C_VEL
